gfCNCPoint4[16844] = {X 523.9193, Y 49.0767, Z -5.5000, A 0.000, B 0.000, C 0.000 }
gfCNCPoint4[16845] = {X 523.4026, Y 49.7085, Z -5.5000, A 0.000, B 0.000, C 0.000 }
gfCNCPoint4[16846] = {X 522.7743, Y 50.2295, Z -5.5000, A 0.000, B 0.000, C 0.000 }
gfCNCPoint4[16847] = {X 522.0579, Y 50.6204, Z -5.5000, A 0.000, B 0.000, C 0.000 }
gfCNCPoint4[16848] = {X 521.2797, Y 50.8666, Z -5.5000, A 0.000, B 0.000, C 0.000 }
gfCNCPoint4[16849] = {X 520.4688, Y 50.9591, Z -5.5000, A 0.000, B 0.000, C 0.000 }
gfCNCPoint4[16850] = {X 519.7998, Y 50.9591, Z -5.5000, A 0.000, B 0.000, C 0.000 }
gfCNCPoint4[16851] = {X 518.8919, Y 50.8568, Z -5.5000, A 0.000, B 0.000, C 0.000 }
gfCNCPoint4[16852] = {X 518.0295, Y 50.5551, Z -5.5000, A 0.000, B 0.000, C 0.000 }
gfCNCPoint4[16853] = {X 517.2559, Y 50.0690, Z -5.5000, A 0.000, B 0.000, C 0.000 }
gfCNCPoint4[16854] = {X 516.6099, Y 49.4230, Z -5.5000, A 0.000, B 0.000, C 0.000 }
gfCNCPoint4[16855] = {X 516.1238, Y 48.6494, Z -5.5000, A 0.000, B 0.000, C 0.000 }
gfCNCPoint4[16856] = {X 515.8221, Y 47.7870, Z -5.5000, A 0.000, B 0.000, C 0.000 }
gfCNCPoint4[16857] = {X 515.7198, Y 46.8791, Z -5.5000, A 0.000, B 0.000, C 0.000 }
gfCNCPoint4[16858] = {X 515.7198, Y 39.9011, Z -5.5000, A 0.000, B 0.000, C 0.000 }
gfCNCPoint4[16859] = {X 515.8209, Y 38.9982, Z -5.5000, A 0.000, B 0.000, C 0.000 }
gfCNCPoint4[16860] = {X 516.1194, Y 38.1401, Z -5.5000, A 0.000, B 0.000, C 0.000 }
gfCNCPoint4[16861] = {X 516.6003, Y 37.3693, Z -5.5000, A 0.000, B 0.000, C 0.000 }
gfCNCPoint4[16862] = {X 517.2399, Y 36.7241, Z -5.5000, A 0.000, B 0.000, C 0.000 }
gfCNCPoint4[16863] = {X 518.0064, Y 36.2364, Z -5.5000, A 0.000, B 0.000, C 0.000 }
gfCNCPoint4[16864] = {X 518.8619, Y 35.9304, Z -5.5000, A 0.000, B 0.000, C 0.000 }
gfCNCPoint4[16865] = {X 519.7638, Y 35.8213, Z -5.5000, A 0.000, B 0.000, C 0.000 }
gfCNCPoint4[16866] = {X 520.5236, Y 35.8215, Z -5.5000, A 0.000, B 0.000, C 0.000 }
gfCNCPoint4[16867] = {X 521.3288, Y 35.9129, Z -5.5000, A 0.000, B 0.000, C 0.000 }
gfCNCPoint4[16868] = {X 522.1000, Y 36.1617, Z -5.5000, A 0.000, B 0.000, C 0.000 }
gfCNCPoint4[16869] = {X 522.8069, Y 36.5579, Z -5.5000, A 0.000, B 0.000, C 0.000 }
gfCNCPoint4[16870] = {X 523.4215, Y 37.0861, Z -5.5000, A 0.000, B 0.000, C 0.000 }
gfCNCPoint4[16871] = {X 523.9196, Y 37.7253, Z -5.5000, A 0.000, B 0.000, C 0.000 }
gfCNCPoint4[16872] = {X 534.8719, Y 37.7258, Z -5.5000, A 0.000, B 0.000, C 0.000 }
gfCNCPoint4[16873] = {X 534.8719, Y 33.7257, Z -5.5000, A 0.000, B 0.000, C 0.000 }
gfCNCPoint4[16874] = {X 529.9775, Y 33.7254, Z -5.5000, A 0.000, B 0.000, C 0.000 }
gfCNCPoint4[16875] = {X 529.9071, Y 33.8366, Z -5.5000, A 0.000, B 0.000, C 0.000 }
gfCNCPoint4[16876] = {X 529.2612, Y 34.5790, Z -5.5000, A 0.000, B 0.000, C 0.000 }
gfCNCPoint4[16877] = {X 528.4563, Y 35.1452, Z -5.5000, A 0.000, B 0.000, C 0.000 }
gfCNCPoint4[16878] = {X 527.5392, Y 35.5023, Z -5.5000, A 0.000, B 0.000, C 0.000 }
gfCNCPoint4[16879] = {X 526.5634, Y 35.6293, Z -5.5000, A 0.000, B 0.000, C 0.000 }
gfCNCPoint4[16880] = {X 525.8868, Y 35.6295, Z -5.5000, A 0.000, B 0.000, C 0.000 }
gfCNCPoint4[16881] = {X 524.9789, Y 35.5272, Z -5.5000, A 0.000, B 0.000, C 0.000 }
gfCNCPoint4[16882] = {X 524.1165, Y 35.2254, Z -5.5000, A 0.000, B 0.000, C 0.000 }
gfCNCPoint4[16883] = {X 523.3429, Y 34.7393, Z -5.5000, A 0.000, B 0.000, C 0.000 }
gfCNCPoint4[16884] = {X 522.6969, Y 34.0933, Z -5.5000, A 0.000, B 0.000, C 0.000 }
gfCNCPoint4[16885] = {X 522.2108, Y 33.3197, Z -5.5000, A 0.000, B 0.000, C 0.000 }
gfCNCPoint4[16886] = {X 521.9091, Y 32.4573, Z -5.5000, A 0.000, B 0.000, C 0.000 }
gfCNCPoint4[16887] = {X 521.8068, Y 31.5495, Z -5.5000, A 0.000, B 0.000, C 0.000 }
gfCNCPoint4[16888] = {X 521.8068, Y 24.5714, Z -5.5000, A 0.000, B 0.000, C 0.000 }
gfCNCPoint4[16889] = {X 521.9079, Y 23.6684, Z -5.5000, A 0.000, B 0.000, C 0.000 }
gfCNCPoint4[16890] = {X 522.2065, Y 22.8102, Z -5.5000, A 0.000, B 0.000, C 0.000 }
gfCNCPoint4[16891] = {X 522.6876, Y 22.0393, Z -5.5000, A 0.000, B 0.000, C 0.000 }
gfCNCPoint4[16892] = {X 523.3273, Y 21.3940, Z -5.5000, A 0.000, B 0.000, C 0.000 }
gfCNCPoint4[16893] = {X 524.0941, Y 20.9064, Z -5.5000, A 0.000, B 0.000, C 0.000 }
gfCNCPoint4[16894] = {X 524.9497, Y 20.6005, Z -5.5000, A 0.000, B 0.000, C 0.000 }
gfCNCPoint4[16895] = {X 525.8518, Y 20.4916, Z -5.5000, A 0.000, B 0.000, C 0.000 }
gfCNCPoint4[16896] = {X 526.5672, Y 20.4916, Z -5.5000, A 0.000, B 0.000, C 0.000 }
gfCNCPoint4[16897] = {X 527.3709, Y 20.5794, Z -5.5000, A 0.000, B 0.000, C 0.000 }
gfCNCPoint4[16898] = {X 528.1415, Y 20.8238, Z -5.5000, A 0.000, B 0.000, C 0.000 }
gfCNCPoint4[16899] = {X 528.8488, Y 21.2155, Z -5.5000, A 0.000, B 0.000, C 0.000 }
gfCNCPoint4[16900] = {X 529.4649, Y 21.7389, Z -5.5000, A 0.000, B 0.000, C 0.000 }
gfCNCPoint4[16901] = {X 529.9658, Y 22.3735, Z -5.5000, A 0.000, B 0.000, C 0.000 }
gfCNCPoint4[16902] = {X 534.8719, Y 22.3737, Z -5.5000, A 0.000, B 0.000, C 0.000 }
gfCNCPoint4[16903] = {X 534.8719, Y 19.4621, Z -5.5000, A 0.000, B 0.000, C 0.000 }
gfCNCPoint4[16904] = {X 524.0609, Y 19.4619, Z -5.5000, A 0.000, B 0.000, C 0.000 }
gfCNCPoint4[16905] = {X 524.0087, Y 19.5442, Z -5.5000, A 0.000, B 0.000, C 0.000 }
gfCNCPoint4[16906] = {X 523.5061, Y 20.1604, Z -5.5000, A 0.000, B 0.000, C 0.000 }
gfCNCPoint4[16907] = {X 522.8935, Y 20.6674, Z -5.5000, A 0.000, B 0.000, C 0.000 }
gfCNCPoint4[16908] = {X 522.1942, Y 21.0459, Z -5.5000, A 0.000, B 0.000, C 0.000 }
gfCNCPoint4[16909] = {X 521.4348, Y 21.2816, Z -5.5000, A 0.000, B 0.000, C 0.000 }
gfCNCPoint4[16910] = {X 520.6440, Y 21.3656, Z -5.5000, A 0.000, B 0.000, C 0.000 }
gfCNCPoint4[16911] = {X 519.9691, Y 21.3657, Z -5.5000, A 0.000, B 0.000, C 0.000 }
gfCNCPoint4[16912] = {X 519.0612, Y 21.2634, Z -5.5000, A 0.000, B 0.000, C 0.000 }
gfCNCPoint4[16913] = {X 518.1989, Y 20.9617, Z -5.5000, A 0.000, B 0.000, C 0.000 }
gfCNCPoint4[16914] = {X 517.4253, Y 20.4756, Z -5.5000, A 0.000, B 0.000, C 0.000 }
gfCNCPoint4[16915] = {X 516.7792, Y 19.8296, Z -5.5000, A 0.000, B 0.000, C 0.000 }
gfCNCPoint4[16916] = {X 516.2932, Y 19.0560, Z -5.5000, A 0.000, B 0.000, C 0.000 }
gfCNCPoint4[16917] = {X 515.9914, Y 18.1936, Z -5.5000, A 0.000, B 0.000, C 0.000 }
gfCNCPoint4[16918] = {X 515.8891, Y 17.2857, Z -5.5000, A 0.000, B 0.000, C 0.000 }
gfCNCPoint4[16919] = {X 515.8891, Y 10.3077, Z -5.5000, A 0.000, B 0.000, C 0.000 }
gfCNCPoint4[16920] = {X 515.9902, Y 9.4050, Z -5.5000, A 0.000, B 0.000, C 0.000 }
gfCNCPoint4[16921] = {X 516.2885, Y 8.5471, Z -5.5000, A 0.000, B 0.000, C 0.000 }
gfCNCPoint4[16922] = {X 516.7693, Y 7.7764, Z -5.5000, A 0.000, B 0.000, C 0.000 }
gfCNCPoint4[16923] = {X 517.4086, Y 7.1312, Z -5.5000, A 0.000, B 0.000, C 0.000 }
gfCNCPoint4[16924] = {X 518.1749, Y 6.6434, Z -5.5000, A 0.000, B 0.000, C 0.000 }
gfCNCPoint4[16925] = {X 519.0301, Y 6.3372, Z -5.5000, A 0.000, B 0.000, C 0.000 }
gfCNCPoint4[16926] = {X 519.9318, Y 6.2279, Z -5.5000, A 0.000, B 0.000, C 0.000 }
gfCNCPoint4[16927] = {X 520.6480, Y 6.2279, Z -5.5000, A 0.000, B 0.000, C 0.000 }
gfCNCPoint4[16928] = {X 521.4520, Y 6.3154, Z -5.5000, A 0.000, B 0.000, C 0.000 }
gfCNCPoint4[16929] = {X 522.2230, Y 6.5597, Z -5.5000, A 0.000, B 0.000, C 0.000 }
gfCNCPoint4[16930] = {X 522.9306, Y 6.9514, Z -5.5000, A 0.000, B 0.000, C 0.000 }
gfCNCPoint4[16931] = {X 523.5471, Y 7.4750, Z -5.5000, A 0.000, B 0.000, C 0.000 }
gfCNCPoint4[16932] = {X 524.0482, Y 8.1098, Z -5.5000, A 0.000, B 0.000, C 0.000 }
gfCNCPoint4[16933] = {X 533.9635, Y 8.1100, Z -5.5000, A 0.000, B 0.000, C 0.000 }
gfCNCPoint4[16934] = {X 533.9636, Y 4.1100, Z -5.5000, A 0.000, B 0.000, C 0.000 }
gfCNCPoint4[16935] = {X 533.9635, Y 8.1900, Z -5.5000, A 0.000, B 0.000, C 0.000 }
gfCNCPoint4[16936] = {X 543.7544, Y 8.1902, Z -5.5000, A 0.000, B 0.000, C 0.000 }
gfCNCPoint4[16937] = {X 544.6628, Y 8.2686, Z -5.5000, A 0.000, B 0.000, C 0.000 }
gfCNCPoint4[16938] = {X 545.5299, Y 8.5504, Z -5.5000, A 0.000, B 0.000, C 0.000 }
gfCNCPoint4[16939] = {X 546.3109, Y 9.0210, Z -5.5000, A 0.000, B 0.000, C 0.000 }
gfCNCPoint4[16940] = {X 546.9651, Y 9.6561, Z -5.5000, A 0.000, B 0.000, C 0.000 }
gfCNCPoint4[16941] = {X 547.4587, Y 10.4228, Z -5.5000, A 0.000, B 0.000, C 0.000 }
gfCNCPoint4[16942] = {X 547.7661, Y 11.2812, Z -5.5000, A 0.000, B 0.000, C 0.000 }
gfCNCPoint4[16943] = {X 547.8714, Y 12.1868, Z -5.5000, A 0.000, B 0.000, C 0.000 }
gfCNCPoint4[16944] = {X 547.8712, Y 13.0192, Z -5.5000, A 0.000, B 0.000, C 0.000 }
gfCNCPoint4[16945] = {X 547.7627, Y 13.9043, Z -5.5000, A 0.000, B 0.000, C 0.000 }
gfCNCPoint4[16946] = {X 547.4608, Y 14.7433, Z -5.5000, A 0.000, B 0.000, C 0.000 }
gfCNCPoint4[16947] = {X 546.9806, Y 15.4946, Z -5.5000, A 0.000, B 0.000, C 0.000 }
gfCNCPoint4[16948] = {X 546.3458, Y 16.1209, Z -5.5000, A 0.000, B 0.000, C 0.000 }
gfCNCPoint4[16949] = {X 546.3444, Y 41.0656, Z -5.5000, A 0.000, B 0.000, C 0.000 }
gfCNCPoint4[16950] = {X 546.4832, Y 41.1792, Z -5.5000, A 0.000, B 0.000, C 0.000 }
gfCNCPoint4[16951] = {X 547.0690, Y 41.8056, Z -5.5000, A 0.000, B 0.000, C 0.000 }
gfCNCPoint4[16952] = {X 547.5079, Y 42.5426, Z -5.5000, A 0.000, B 0.000, C 0.000 }
gfCNCPoint4[16953] = {X 547.7795, Y 43.3561, Z -5.5000, A 0.000, B 0.000, C 0.000 }
gfCNCPoint4[16954] = {X 547.8714, Y 44.2089, Z -5.5000, A 0.000, B 0.000, C 0.000 }
gfCNCPoint4[16955] = {X 547.8714, Y 45.0000, Z -5.5000, A 0.000, B 0.000, C 0.000 }
gfCNCPoint4[16956] = {X 547.7662, Y 45.9056, Z -5.5000, A 0.000, B 0.000, C 0.000 }
gfCNCPoint4[16957] = {X 547.4587, Y 46.7640, Z -5.5000, A 0.000, B 0.000, C 0.000 }
gfCNCPoint4[16958] = {X 546.9651, Y 47.5306, Z -5.5000, A 0.000, B 0.000, C 0.000 }
gfCNCPoint4[16959] = {X 546.3109, Y 48.1657, Z -5.5000, A 0.000, B 0.000, C 0.000 }
gfCNCPoint4[16960] = {X 545.5299, Y 48.6363, Z -5.5000, A 0.000, B 0.000, C 0.000 }
gfCNCPoint4[16961] = {X 544.6628, Y 48.9180, Z -5.5000, A 0.000, B 0.000, C 0.000 }
gfCNCPoint4[16962] = {X 543.7544, Y 48.9963, Z -5.5000, A 0.000, B 0.000, C 0.000 }
gfCNCPoint4[16963] = {X 523.8762, Y 48.9967, Z -5.5000, A 0.000, B 0.000, C 0.000 }
gfCNCPoint4[16964] = {X 523.3698, Y 49.6277, Z -5.5000, A 0.000, B 0.000, C 0.000 }
gfCNCPoint4[16965] = {X 522.7508, Y 50.1487, Z -5.5000, A 0.000, B 0.000, C 0.000 }
gfCNCPoint4[16966] = {X 522.0425, Y 50.5399, Z -5.5000, A 0.000, B 0.000, C 0.000 }
gfCNCPoint4[16967] = {X 521.2719, Y 50.7865, Z -5.5000, A 0.000, B 0.000, C 0.000 }
gfCNCPoint4[16968] = {X 520.4681, Y 50.8791, Z -5.5000, A 0.000, B 0.000, C 0.000 }
gfCNCPoint4[16969] = {X 519.7998, Y 50.8791, Z -5.5000, A 0.000, B 0.000, C 0.000 }
gfCNCPoint4[16970] = {X 518.9097, Y 50.7788, Z -5.5000, A 0.000, B 0.000, C 0.000 }
gfCNCPoint4[16971] = {X 518.0642, Y 50.4830, Z -5.5000, A 0.000, B 0.000, C 0.000 }
gfCNCPoint4[16972] = {X 517.3058, Y 50.0064, Z -5.5000, A 0.000, B 0.000, C 0.000 }
gfCNCPoint4[16973] = {X 516.6724, Y 49.3731, Z -5.5000, A 0.000, B 0.000, C 0.000 }
gfCNCPoint4[16974] = {X 516.1959, Y 48.6147, Z -5.5000, A 0.000, B 0.000, C 0.000 }
gfCNCPoint4[16975] = {X 515.9001, Y 47.7692, Z -5.5000, A 0.000, B 0.000, C 0.000 }
gfCNCPoint4[16976] = {X 515.7998, Y 46.8791, Z -5.5000, A 0.000, B 0.000, C 0.000 }
gfCNCPoint4[16977] = {X 515.7998, Y 39.9011, Z -5.5000, A 0.000, B 0.000, C 0.000 }
gfCNCPoint4[16978] = {X 515.9001, Y 39.0110, Z -5.5000, A 0.000, B 0.000, C 0.000 }
gfCNCPoint4[16979] = {X 516.1959, Y 38.1655, Z -5.5000, A 0.000, B 0.000, C 0.000 }
gfCNCPoint4[16980] = {X 516.6725, Y 37.4071, Z -5.5000, A 0.000, B 0.000, C 0.000 }
gfCNCPoint4[16981] = {X 517.3058, Y 36.7738, Z -5.5000, A 0.000, B 0.000, C 0.000 }
gfCNCPoint4[16982] = {X 518.0643, Y 36.2972, Z -5.5000, A 0.000, B 0.000, C 0.000 }
gfCNCPoint4[16983] = {X 518.9097, Y 36.0014, Z -5.5000, A 0.000, B 0.000, C 0.000 }
gfCNCPoint4[16984] = {X 519.7998, Y 35.9011, Z -5.5000, A 0.000, B 0.000, C 0.000 }
gfCNCPoint4[16985] = {X 520.5225, Y 35.9015, Z -5.5000, A 0.000, B 0.000, C 0.000 }
gfCNCPoint4[16986] = {X 521.3205, Y 35.9930, Z -5.5000, A 0.000, B 0.000, C 0.000 }
gfCNCPoint4[16987] = {X 522.0842, Y 36.2421, Z -5.5000, A 0.000, B 0.000, C 0.000 }
gfCNCPoint4[16988] = {X 522.7826, Y 36.6387, Z -5.5000, A 0.000, B 0.000, C 0.000 }
gfCNCPoint4[16989] = {X 523.3878, Y 37.1669, Z -5.5000, A 0.000, B 0.000, C 0.000 }
gfCNCPoint4[16990] = {X 523.8752, Y 37.8053, Z -5.5000, A 0.000, B 0.000, C 0.000 }
gfCNCPoint4[16991] = {X 534.9519, Y 37.8058, Z -5.5000, A 0.000, B 0.000, C 0.000 }
gfCNCPoint4[16992] = {X 534.9519, Y 34.0457, Z -5.5000, A 0.000, B 0.000, C 0.000 }
gfCNCPoint4[16993] = {X 534.9521, Y 33.6457, Z -5.5000, A 0.000, B 0.000, C 0.000 }
gfCNCPoint4[16994] = {X 529.9335, Y 33.6454, Z -5.5000, A 0.000, B 0.000, C 0.000 }
gfCNCPoint4[16995] = {X 529.8226, Y 33.8185, Z -5.5000, A 0.000, B 0.000, C 0.000 }
gfCNCPoint4[16996] = {X 529.1831, Y 34.5416, Z -5.5000, A 0.000, B 0.000, C 0.000 }
gfCNCPoint4[16997] = {X 528.3890, Y 35.0904, Z -5.5000, A 0.000, B 0.000, C 0.000 }
gfCNCPoint4[16998] = {X 527.4865, Y 35.4330, Z -5.5000, A 0.000, B 0.000, C 0.000 }
gfCNCPoint4[16999] = {X 526.5283, Y 35.5495, Z -5.5000, A 0.000, B 0.000, C 0.000 }
gfCNCPoint4[17000] = {X 525.8868, Y 35.5495, Z -5.5000, A 0.000, B 0.000, C 0.000 }
gfCNCPoint4[17001] = {X 524.9967, Y 35.4492, Z -5.5000, A 0.000, B 0.000, C 0.000 }
gfCNCPoint4[17002] = {X 524.1512, Y 35.1533, Z -5.5000, A 0.000, B 0.000, C 0.000 }
gfCNCPoint4[17003] = {X 523.3928, Y 34.6768, Z -5.5000, A 0.000, B 0.000, C 0.000 }
gfCNCPoint4[17004] = {X 522.7594, Y 34.0434, Z -5.5000, A 0.000, B 0.000, C 0.000 }
gfCNCPoint4[17005] = {X 522.2829, Y 33.2850, Z -5.5000, A 0.000, B 0.000, C 0.000 }
gfCNCPoint4[17006] = {X 521.9870, Y 32.4395, Z -5.5000, A 0.000, B 0.000, C 0.000 }
gfCNCPoint4[17007] = {X 521.8868, Y 31.5495, Z -5.5000, A 0.000, B 0.000, C 0.000 }
gfCNCPoint4[17008] = {X 521.8868, Y 24.5714, Z -5.5000, A 0.000, B 0.000, C 0.000 }
gfCNCPoint4[17009] = {X 521.9870, Y 23.6813, Z -5.5000, A 0.000, B 0.000, C 0.000 }
gfCNCPoint4[17010] = {X 522.2829, Y 22.8359, Z -5.5000, A 0.000, B 0.000, C 0.000 }
gfCNCPoint4[17011] = {X 522.7594, Y 22.0775, Z -5.5000, A 0.000, B 0.000, C 0.000 }
gfCNCPoint4[17012] = {X 523.3928, Y 21.4441, Z -5.5000, A 0.000, B 0.000, C 0.000 }
gfCNCPoint4[17013] = {X 524.1512, Y 20.9675, Z -5.5000, A 0.000, B 0.000, C 0.000 }
gfCNCPoint4[17014] = {X 524.9967, Y 20.6717, Z -5.5000, A 0.000, B 0.000, C 0.000 }
gfCNCPoint4[17015] = {X 525.8868, Y 20.5714, Z -5.5000, A 0.000, B 0.000, C 0.000 }
gfCNCPoint4[17016] = {X 526.5664, Y 20.5716, Z -5.5000, A 0.000, B 0.000, C 0.000 }
gfCNCPoint4[17017] = {X 527.3629, Y 20.6594, Z -5.5000, A 0.000, B 0.000, C 0.000 }
gfCNCPoint4[17018] = {X 528.1259, Y 20.9043, Z -5.5000, A 0.000, B 0.000, C 0.000 }
gfCNCPoint4[17019] = {X 528.8248, Y 21.2962, Z -5.5000, A 0.000, B 0.000, C 0.000 }
gfCNCPoint4[17020] = {X 529.4315, Y 21.8197, Z -5.5000, A 0.000, B 0.000, C 0.000 }
gfCNCPoint4[17021] = {X 529.9217, Y 22.4535, Z -5.5000, A 0.000, B 0.000, C 0.000 }
gfCNCPoint4[17022] = {X 534.9519, Y 22.4537, Z -5.5000, A 0.000, B 0.000, C 0.000 }
gfCNCPoint4[17023] = {X 534.9519, Y 19.7821, Z -5.5000, A 0.000, B 0.000, C 0.000 }
gfCNCPoint4[17024] = {X 534.9522, Y 19.3821, Z -5.5000, A 0.000, B 0.000, C 0.000 }
gfCNCPoint4[17025] = {X 524.0169, Y 19.3819, Z -5.5000, A 0.000, B 0.000, C 0.000 }
gfCNCPoint4[17026] = {X 523.9048, Y 19.5550, Z -5.5000, A 0.000, B 0.000, C 0.000 }
gfCNCPoint4[17027] = {X 523.2653, Y 20.2779, Z -5.5000, A 0.000, B 0.000, C 0.000 }
gfCNCPoint4[17028] = {X 522.4713, Y 20.8267, Z -5.5000, A 0.000, B 0.000, C 0.000 }
gfCNCPoint4[17029] = {X 521.5689, Y 21.1693, Z -5.5000, A 0.000, B 0.000, C 0.000 }
gfCNCPoint4[17030] = {X 520.6107, Y 21.2857, Z -5.5000, A 0.000, B 0.000, C 0.000 }
gfCNCPoint4[17031] = {X 519.9691, Y 21.2857, Z -5.5000, A 0.000, B 0.000, C 0.000 }
gfCNCPoint4[17032] = {X 519.0790, Y 21.1854, Z -5.5000, A 0.000, B 0.000, C 0.000 }
gfCNCPoint4[17033] = {X 518.2336, Y 20.8896, Z -5.5000, A 0.000, B 0.000, C 0.000 }
gfCNCPoint4[17034] = {X 517.4751, Y 20.4130, Z -5.5000, A 0.000, B 0.000, C 0.000 }
gfCNCPoint4[17035] = {X 516.8418, Y 19.7797, Z -5.5000, A 0.000, B 0.000, C 0.000 }
gfCNCPoint4[17036] = {X 516.3652, Y 19.0212, Z -5.5000, A 0.000, B 0.000, C 0.000 }
gfCNCPoint4[17037] = {X 516.0694, Y 18.1758, Z -5.5000, A 0.000, B 0.000, C 0.000 }
gfCNCPoint4[17038] = {X 515.9691, Y 17.2857, Z -5.5000, A 0.000, B 0.000, C 0.000 }
gfCNCPoint4[17039] = {X 515.9691, Y 10.3077, Z -5.5000, A 0.000, B 0.000, C 0.000 }
gfCNCPoint4[17040] = {X 516.0694, Y 9.4176, Z -5.5000, A 0.000, B 0.000, C 0.000 }
gfCNCPoint4[17041] = {X 516.3652, Y 8.5721, Z -5.5000, A 0.000, B 0.000, C 0.000 }
gfCNCPoint4[17042] = {X 516.8418, Y 7.8137, Z -5.5000, A 0.000, B 0.000, C 0.000 }
gfCNCPoint4[17043] = {X 517.4752, Y 7.1803, Z -5.5000, A 0.000, B 0.000, C 0.000 }
gfCNCPoint4[17044] = {X 518.2336, Y 6.7038, Z -5.5000, A 0.000, B 0.000, C 0.000 }
gfCNCPoint4[17045] = {X 519.0791, Y 6.4080, Z -5.5000, A 0.000, B 0.000, C 0.000 }
gfCNCPoint4[17046] = {X 519.9692, Y 6.3077, Z -5.5000, A 0.000, B 0.000, C 0.000 }
gfCNCPoint4[17047] = {X 520.6472, Y 6.3079, Z -5.5000, A 0.000, B 0.000, C 0.000 }
gfCNCPoint4[17048] = {X 521.4441, Y 6.3955, Z -5.5000, A 0.000, B 0.000, C 0.000 }
gfCNCPoint4[17049] = {X 522.2074, Y 6.6402, Z -5.5000, A 0.000, B 0.000, C 0.000 }
gfCNCPoint4[17050] = {X 522.9066, Y 7.0322, Z -5.5000, A 0.000, B 0.000, C 0.000 }
gfCNCPoint4[17051] = {X 523.5137, Y 7.5557, Z -5.5000, A 0.000, B 0.000, C 0.000 }
gfCNCPoint4[17052] = {X 524.0041, Y 8.1898, Z -5.5000, A 0.000, B 0.000, C 0.000 }
gfCNCPoint4[17053] = {X 533.9635, Y 8.1900, Z -5.5000, A 0.000, B 0.000, C 0.000 }
gfCNCPoint4[17054] = {X 533.9636, Y 4.1100, Z -5.5000, A 0.000, B 0.000, C 0.000 }
gfCNCPoint4[17055] = {X 533.9636, Y 4.1100, Z -2.5000, A 0.000, B 0.000, C 0.000 }
gfCNCPoint4[17056] = {X 533.9636, Y 4.1100, Z 11.0000, A 0.000, B 0.000, C 0.000 }
gfCNCPoint4[17057] = {X 419.6144, Y 26.5282, Z 11.0000, A 0.000, B 0.000, C 0.000 }
gfCNCPoint4[17058] = {X 419.6144, Y 26.5282, Z -2.5000, A 0.000, B 0.000, C 0.000 }
gfCNCPoint4[17059] = {X 419.6144, Y 26.5282, Z -5.5000, A 0.000, B 0.000, C 0.000 }
gfCNCPoint4[17060] = {X 416.1509, Y 24.3717, Z -5.5000, A 0.000, B 0.000, C 0.000 }
gfCNCPoint4[17061] = {X 411.5473, Y 31.7652, Z -5.5000, A 0.000, B 0.000, C 0.000 }
gfCNCPoint4[17062] = {X 411.5479, Y 40.8978, Z -5.5000, A 0.000, B 0.000, C 0.000 }
gfCNCPoint4[17063] = {X 412.1861, Y 41.5837, Z -5.5000, A 0.000, B 0.000, C 0.000 }
gfCNCPoint4[17064] = {X 412.6662, Y 42.3882, Z -5.5000, A 0.000, B 0.000, C 0.000 }
gfCNCPoint4[17065] = {X 412.9668, Y 43.2755, Z -5.5000, A 0.000, B 0.000, C 0.000 }
gfCNCPoint4[17066] = {X 413.0747, Y 44.2062, Z -5.5000, A 0.000, B 0.000, C 0.000 }
gfCNCPoint4[17067] = {X 413.0747, Y 45.0002, Z -5.5000, A 0.000, B 0.000, C 0.000 }
gfCNCPoint4[17068] = {X 412.9663, Y 45.9614, Z -5.5000, A 0.000, B 0.000, C 0.000 }
gfCNCPoint4[17069] = {X 412.6468, Y 46.8745, Z -5.5000, A 0.000, B 0.000, C 0.000 }
gfCNCPoint4[17070] = {X 412.1321, Y 47.6936, Z -5.5000, A 0.000, B 0.000, C 0.000 }
gfCNCPoint4[17071] = {X 411.4481, Y 48.3776, Z -5.5000, A 0.000, B 0.000, C 0.000 }
gfCNCPoint4[17072] = {X 410.6290, Y 48.8922, Z -5.5000, A 0.000, B 0.000, C 0.000 }
gfCNCPoint4[17073] = {X 409.7159, Y 49.2117, Z -5.5000, A 0.000, B 0.000, C 0.000 }
gfCNCPoint4[17074] = {X 408.7547, Y 49.3200, Z -5.5000, A 0.000, B 0.000, C 0.000 }
gfCNCPoint4[17075] = {X 402.3112, Y 49.3200, Z -5.5000, A 0.000, B 0.000, C 0.000 }
gfCNCPoint4[17076] = {X 401.3546, Y 49.2127, Z -5.5000, A 0.000, B 0.000, C 0.000 }
gfCNCPoint4[17077] = {X 400.4455, Y 48.8963, Z -5.5000, A 0.000, B 0.000, C 0.000 }
gfCNCPoint4[17078] = {X 399.6290, Y 48.3864, Z -5.5000, A 0.000, B 0.000, C 0.000 }
gfCNCPoint4[17079] = {X 398.9457, Y 47.7084, Z -5.5000, A 0.000, B 0.000, C 0.000 }
gfCNCPoint4[17080] = {X 398.4295, Y 46.8959, Z -5.5000, A 0.000, B 0.000, C 0.000 }
gfCNCPoint4[17081] = {X 398.1060, Y 45.9892, Z -5.5000, A 0.000, B 0.000, C 0.000 }
gfCNCPoint4[17082] = {X 397.9913, Y 45.0335, Z -5.5000, A 0.000, B 0.000, C 0.000 }
gfCNCPoint4[17083] = {X 397.9916, Y 44.1528, Z -5.5000, A 0.000, B 0.000, C 0.000 }
gfCNCPoint4[17084] = {X 398.1015, Y 43.2391, Z -5.5000, A 0.000, B 0.000, C 0.000 }
gfCNCPoint4[17085] = {X 398.4024, Y 42.3694, Z -5.5000, A 0.000, B 0.000, C 0.000 }
gfCNCPoint4[17086] = {X 398.8807, Y 41.5832, Z -5.5000, A 0.000, B 0.000, C 0.000 }
gfCNCPoint4[17087] = {X 399.5147, Y 40.9161, Z -5.5000, A 0.000, B 0.000, C 0.000 }
gfCNCPoint4[17088] = {X 399.4729, Y 31.6010, Z -5.5000, A 0.000, B 0.000, C 0.000 }
gfCNCPoint4[17089] = {X 393.5178, Y 21.2453, Z -5.5000, A 0.000, B 0.000, C 0.000 }
gfCNCPoint4[17090] = {X 392.6297, Y 19.7345, Z -5.5000, A 0.000, B 0.000, C 0.000 }
gfCNCPoint4[17091] = {X 391.7131, Y 18.2409, Z -5.5000, A 0.000, B 0.000, C 0.000 }
gfCNCPoint4[17092] = {X 391.2305, Y 17.5698, Z -5.5000, A 0.000, B 0.000, C 0.000 }
gfCNCPoint4[17093] = {X 390.6669, Y 16.9652, Z -5.5000, A 0.000, B 0.000, C 0.000 }
gfCNCPoint4[17094] = {X 389.7902, Y 16.4728, Z -5.5000, A 0.000, B 0.000, C 0.000 }
gfCNCPoint4[17095] = {X 389.0510, Y 15.7911, Z -5.5000, A 0.000, B 0.000, C 0.000 }
gfCNCPoint4[17096] = {X 388.4895, Y 14.9569, Z -5.5000, A 0.000, B 0.000, C 0.000 }
gfCNCPoint4[17097] = {X 388.1361, Y 14.0156, Z -5.5000, A 0.000, B 0.000, C 0.000 }
gfCNCPoint4[17098] = {X 388.0098, Y 13.0180, Z -5.5000, A 0.000, B 0.000, C 0.000 }
gfCNCPoint4[17099] = {X 388.0096, Y 12.1868, Z -5.5000, A 0.000, B 0.000, C 0.000 }
gfCNCPoint4[17100] = {X 388.1179, Y 11.2255, Z -5.5000, A 0.000, B 0.000, C 0.000 }
gfCNCPoint4[17101] = {X 388.4374, Y 10.3125, Z -5.5000, A 0.000, B 0.000, C 0.000 }
gfCNCPoint4[17102] = {X 388.9521, Y 9.4933, Z -5.5000, A 0.000, B 0.000, C 0.000 }
gfCNCPoint4[17103] = {X 389.6361, Y 8.8093, Z -5.5000, A 0.000, B 0.000, C 0.000 }
gfCNCPoint4[17104] = {X 390.4552, Y 8.2946, Z -5.5000, A 0.000, B 0.000, C 0.000 }
gfCNCPoint4[17105] = {X 391.3683, Y 7.9751, Z -5.5000, A 0.000, B 0.000, C 0.000 }
gfCNCPoint4[17106] = {X 392.3296, Y 7.8668, Z -5.5000, A 0.000, B 0.000, C 0.000 }
gfCNCPoint4[17107] = {X 399.1118, Y 7.8668, Z -5.5000, A 0.000, B 0.000, C 0.000 }
gfCNCPoint4[17108] = {X 400.0730, Y 7.9751, Z -5.5000, A 0.000, B 0.000, C 0.000 }
gfCNCPoint4[17109] = {X 400.9861, Y 8.2946, Z -5.5000, A 0.000, B 0.000, C 0.000 }
gfCNCPoint4[17110] = {X 401.8052, Y 8.8093, Z -5.5000, A 0.000, B 0.000, C 0.000 }
gfCNCPoint4[17111] = {X 402.4893, Y 9.4933, Z -5.5000, A 0.000, B 0.000, C 0.000 }
gfCNCPoint4[17112] = {X 403.0039, Y 10.3124, Z -5.5000, A 0.000, B 0.000, C 0.000 }
gfCNCPoint4[17113] = {X 403.3234, Y 11.2255, Z -5.5000, A 0.000, B 0.000, C 0.000 }
gfCNCPoint4[17114] = {X 403.4318, Y 12.1868, Z -5.5000, A 0.000, B 0.000, C 0.000 }
gfCNCPoint4[17115] = {X 403.4318, Y 12.9782, Z -5.5000, A 0.000, B 0.000, C 0.000 }
gfCNCPoint4[17116] = {X 403.3293, Y 13.9134, Z -5.5000, A 0.000, B 0.000, C 0.000 }
gfCNCPoint4[17117] = {X 403.0267, Y 14.8043, Z -5.5000, A 0.000, B 0.000, C 0.000 }
gfCNCPoint4[17118] = {X 405.3561, Y 18.8228, Z -5.5000, A 0.000, B 0.000, C 0.000 }
gfCNCPoint4[17119] = {X 407.8733, Y 14.7536, Z -5.5000, A 0.000, B 0.000, C 0.000 }
gfCNCPoint4[17120] = {X 407.5920, Y 13.9042, Z -5.5000, A 0.000, B 0.000, C 0.000 }
gfCNCPoint4[17121] = {X 407.4917, Y 13.0151, Z -5.5000, A 0.000, B 0.000, C 0.000 }
gfCNCPoint4[17122] = {X 407.4915, Y 12.1868, Z -5.5000, A 0.000, B 0.000, C 0.000 }
gfCNCPoint4[17123] = {X 407.5999, Y 11.2255, Z -5.5000, A 0.000, B 0.000, C 0.000 }
gfCNCPoint4[17124] = {X 407.9194, Y 10.3124, Z -5.5000, A 0.000, B 0.000, C 0.000 }
gfCNCPoint4[17125] = {X 408.4340, Y 9.4933, Z -5.5000, A 0.000, B 0.000, C 0.000 }
gfCNCPoint4[17126] = {X 409.1181, Y 8.8093, Z -5.5000, A 0.000, B 0.000, C 0.000 }
gfCNCPoint4[17127] = {X 409.9372, Y 8.2946, Z -5.5000, A 0.000, B 0.000, C 0.000 }
gfCNCPoint4[17128] = {X 410.8502, Y 7.9751, Z -5.5000, A 0.000, B 0.000, C 0.000 }
gfCNCPoint4[17129] = {X 411.8115, Y 7.8668, Z -5.5000, A 0.000, B 0.000, C 0.000 }
gfCNCPoint4[17130] = {X 419.3245, Y 7.8668, Z -5.5000, A 0.000, B 0.000, C 0.000 }
gfCNCPoint4[17131] = {X 420.2858, Y 7.9751, Z -5.5000, A 0.000, B 0.000, C 0.000 }
gfCNCPoint4[17132] = {X 421.1988, Y 8.2946, Z -5.5000, A 0.000, B 0.000, C 0.000 }
gfCNCPoint4[17133] = {X 422.0179, Y 8.8093, Z -5.5000, A 0.000, B 0.000, C 0.000 }
gfCNCPoint4[17134] = {X 422.7020, Y 9.4933, Z -5.5000, A 0.000, B 0.000, C 0.000 }
gfCNCPoint4[17135] = {X 423.2166, Y 10.3124, Z -5.5000, A 0.000, B 0.000, C 0.000 }
gfCNCPoint4[17136] = {X 423.5361, Y 11.2255, Z -5.5000, A 0.000, B 0.000, C 0.000 }
gfCNCPoint4[17137] = {X 423.6445, Y 12.1868, Z -5.5000, A 0.000, B 0.000, C 0.000 }
gfCNCPoint4[17138] = {X 423.6445, Y 12.9802, Z -5.5000, A 0.000, B 0.000, C 0.000 }
gfCNCPoint4[17139] = {X 423.5517, Y 13.8468, Z -5.5000, A 0.000, B 0.000, C 0.000 }
gfCNCPoint4[17140] = {X 423.2893, Y 14.6779, Z -5.5000, A 0.000, B 0.000, C 0.000 }
gfCNCPoint4[17141] = {X 422.8676, Y 15.4406, Z -5.5000, A 0.000, B 0.000, C 0.000 }
gfCNCPoint4[17142] = {X 422.3034, Y 16.1048, Z -5.5000, A 0.000, B 0.000, C 0.000 }
gfCNCPoint4[17143] = {X 421.6189, Y 16.6442, Z -5.5000, A 0.000, B 0.000, C 0.000 }
gfCNCPoint4[17144] = {X 420.8412, Y 17.0376, Z -5.5000, A 0.000, B 0.000, C 0.000 }
gfCNCPoint4[17145] = {X 420.1248, Y 18.0010, Z -5.5000, A 0.000, B 0.000, C 0.000 }
gfCNCPoint4[17146] = {X 419.4766, Y 19.0115, Z -5.5000, A 0.000, B 0.000, C 0.000 }
gfCNCPoint4[17147] = {X 417.9942, Y 21.4114, Z -5.5000, A 0.000, B 0.000, C 0.000 }
gfCNCPoint4[17148] = {X 416.1509, Y 24.3717, Z -5.5000, A 0.000, B 0.000, C 0.000 }
gfCNCPoint4[17149] = {X 419.5465, Y 26.4860, Z -5.5000, A 0.000, B 0.000, C 0.000 }
gfCNCPoint4[17150] = {X 416.0830, Y 24.3294, Z -5.5000, A 0.000, B 0.000, C 0.000 }
gfCNCPoint4[17151] = {X 411.4673, Y 31.7423, Z -5.5000, A 0.000, B 0.000, C 0.000 }
gfCNCPoint4[17152] = {X 411.4679, Y 40.9345, Z -5.5000, A 0.000, B 0.000, C 0.000 }
gfCNCPoint4[17153] = {X 412.1057, Y 41.6100, Z -5.5000, A 0.000, B 0.000, C 0.000 }
gfCNCPoint4[17154] = {X 412.5859, Y 42.4052, Z -5.5000, A 0.000, B 0.000, C 0.000 }
gfCNCPoint4[17155] = {X 412.8868, Y 43.2842, Z -5.5000, A 0.000, B 0.000, C 0.000 }
gfCNCPoint4[17156] = {X 412.9947, Y 44.2069, Z -5.5000, A 0.000, B 0.000, C 0.000 }
gfCNCPoint4[17157] = {X 412.9947, Y 45.0002, Z -5.5000, A 0.000, B 0.000, C 0.000 }
gfCNCPoint4[17158] = {X 412.8883, Y 45.9436, Z -5.5000, A 0.000, B 0.000, C 0.000 }
gfCNCPoint4[17159] = {X 412.5747, Y 46.8398, Z -5.5000, A 0.000, B 0.000, C 0.000 }
gfCNCPoint4[17160] = {X 412.0696, Y 47.6437, Z -5.5000, A 0.000, B 0.000, C 0.000 }
gfCNCPoint4[17161] = {X 411.3982, Y 48.3150, Z -5.5000, A 0.000, B 0.000, C 0.000 }
gfCNCPoint4[17162] = {X 410.5943, Y 48.8201, Z -5.5000, A 0.000, B 0.000, C 0.000 }
gfCNCPoint4[17163] = {X 409.6981, Y 49.1337, Z -5.5000, A 0.000, B 0.000, C 0.000 }
gfCNCPoint4[17164] = {X 408.7547, Y 49.2400, Z -5.5000, A 0.000, B 0.000, C 0.000 }
gfCNCPoint4[17165] = {X 402.3112, Y 49.2400, Z -5.5000, A 0.000, B 0.000, C 0.000 }
gfCNCPoint4[17166] = {X 401.3723, Y 49.1347, Z -5.5000, A 0.000, B 0.000, C 0.000 }
gfCNCPoint4[17167] = {X 400.4800, Y 48.8242, Z -5.5000, A 0.000, B 0.000, C 0.000 }
gfCNCPoint4[17168] = {X 399.6786, Y 48.3237, Z -5.5000, A 0.000, B 0.000, C 0.000 }
gfCNCPoint4[17169] = {X 399.0080, Y 47.6582, Z -5.5000, A 0.000, B 0.000, C 0.000 }
gfCNCPoint4[17170] = {X 398.5013, Y 46.8608, Z -5.5000, A 0.000, B 0.000, C 0.000 }
gfCNCPoint4[17171] = {X 398.1839, Y 45.9709, Z -5.5000, A 0.000, B 0.000, C 0.000 }
gfCNCPoint4[17172] = {X 398.0713, Y 45.0329, Z -5.5000, A 0.000, B 0.000, C 0.000 }
gfCNCPoint4[17173] = {X 398.0716, Y 44.1538, Z -5.5000, A 0.000, B 0.000, C 0.000 }
gfCNCPoint4[17174] = {X 398.1815, Y 43.2480, Z -5.5000, A 0.000, B 0.000, C 0.000 }
gfCNCPoint4[17175] = {X 398.4827, Y 42.3867, Z -5.5000, A 0.000, B 0.000, C 0.000 }
gfCNCPoint4[17176] = {X 398.9612, Y 41.6098, Z -5.5000, A 0.000, B 0.000, C 0.000 }
gfCNCPoint4[17177] = {X 399.5948, Y 40.9532, Z -5.5000, A 0.000, B 0.000, C 0.000 }
gfCNCPoint4[17178] = {X 399.5528, Y 31.5795, Z -5.5000, A 0.000, B 0.000, C 0.000 }
gfCNCPoint4[17179] = {X 393.5872, Y 21.2054, Z -5.5000, A 0.000, B 0.000, C 0.000 }
gfCNCPoint4[17180] = {X 392.6983, Y 19.6933, Z -5.5000, A 0.000, B 0.000, C 0.000 }
gfCNCPoint4[17181] = {X 391.7809, Y 18.1984, Z -5.5000, A 0.000, B 0.000, C 0.000 }
gfCNCPoint4[17182] = {X 391.2877, Y 17.5134, Z -5.5000, A 0.000, B 0.000, C 0.000 }
gfCNCPoint4[17183] = {X 390.7111, Y 16.8969, Z -5.5000, A 0.000, B 0.000, C 0.000 }
gfCNCPoint4[17184] = {X 389.8466, Y 16.4149, Z -5.5000, A 0.000, B 0.000, C 0.000 }
gfCNCPoint4[17185] = {X 389.1174, Y 15.7456, Z -5.5000, A 0.000, B 0.000, C 0.000 }
gfCNCPoint4[17186] = {X 388.5633, Y 14.9255, Z -5.5000, A 0.000, B 0.000, C 0.000 }
gfCNCPoint4[17187] = {X 388.2144, Y 13.9992, Z -5.5000, A 0.000, B 0.000, C 0.000 }
gfCNCPoint4[17188] = {X 388.0898, Y 13.0173, Z -5.5000, A 0.000, B 0.000, C 0.000 }
gfCNCPoint4[17189] = {X 388.0896, Y 12.1868, Z -5.5000, A 0.000, B 0.000, C 0.000 }
gfCNCPoint4[17190] = {X 388.1959, Y 11.2433, Z -5.5000, A 0.000, B 0.000, C 0.000 }
gfCNCPoint4[17191] = {X 388.5095, Y 10.3472, Z -5.5000, A 0.000, B 0.000, C 0.000 }
gfCNCPoint4[17192] = {X 389.0147, Y 9.5432, Z -5.5000, A 0.000, B 0.000, C 0.000 }
gfCNCPoint4[17193] = {X 389.6860, Y 8.8719, Z -5.5000, A 0.000, B 0.000, C 0.000 }
gfCNCPoint4[17194] = {X 390.4900, Y 8.3667, Z -5.5000, A 0.000, B 0.000, C 0.000 }
gfCNCPoint4[17195] = {X 391.3861, Y 8.0531, Z -5.5000, A 0.000, B 0.000, C 0.000 }
gfCNCPoint4[17196] = {X 392.3296, Y 7.9468, Z -5.5000, A 0.000, B 0.000, C 0.000 }
gfCNCPoint4[17197] = {X 399.1118, Y 7.9468, Z -5.5000, A 0.000, B 0.000, C 0.000 }
gfCNCPoint4[17198] = {X 400.0552, Y 8.0531, Z -5.5000, A 0.000, B 0.000, C 0.000 }
gfCNCPoint4[17199] = {X 400.9514, Y 8.3667, Z -5.5000, A 0.000, B 0.000, C 0.000 }
gfCNCPoint4[17200] = {X 401.7554, Y 8.8718, Z -5.5000, A 0.000, B 0.000, C 0.000 }
gfCNCPoint4[17201] = {X 402.4267, Y 9.5432, Z -5.5000, A 0.000, B 0.000, C 0.000 }
gfCNCPoint4[17202] = {X 402.9319, Y 10.3471, Z -5.5000, A 0.000, B 0.000, C 0.000 }
gfCNCPoint4[17203] = {X 403.2455, Y 11.2433, Z -5.5000, A 0.000, B 0.000, C 0.000 }
gfCNCPoint4[17204] = {X 403.3518, Y 12.1868, Z -5.5000, A 0.000, B 0.000, C 0.000 }
gfCNCPoint4[17205] = {X 403.3518, Y 12.9782, Z -5.5000, A 0.000, B 0.000, C 0.000 }
gfCNCPoint4[17206] = {X 403.2466, Y 13.9164, Z -5.5000, A 0.000, B 0.000, C 0.000 }
gfCNCPoint4[17207] = {X 402.9364, Y 14.8081, Z -5.5000, A 0.000, B 0.000, C 0.000 }
gfCNCPoint4[17208] = {X 405.3539, Y 18.9785, Z -5.5000, A 0.000, B 0.000, C 0.000 }
gfCNCPoint4[17209] = {X 407.9639, Y 14.7593, Z -5.5000, A 0.000, B 0.000, C 0.000 }
gfCNCPoint4[17210] = {X 407.6747, Y 13.9078, Z -5.5000, A 0.000, B 0.000, C 0.000 }
gfCNCPoint4[17211] = {X 407.5717, Y 13.0144, Z -5.5000, A 0.000, B 0.000, C 0.000 }
gfCNCPoint4[17212] = {X 407.5715, Y 12.1868, Z -5.5000, A 0.000, B 0.000, C 0.000 }
gfCNCPoint4[17213] = {X 407.6778, Y 11.2433, Z -5.5000, A 0.000, B 0.000, C 0.000 }
gfCNCPoint4[17214] = {X 407.9914, Y 10.3471, Z -5.5000, A 0.000, B 0.000, C 0.000 }
gfCNCPoint4[17215] = {X 408.4966, Y 9.5432, Z -5.5000, A 0.000, B 0.000, C 0.000 }
gfCNCPoint4[17216] = {X 409.1679, Y 8.8718, Z -5.5000, A 0.000, B 0.000, C 0.000 }
gfCNCPoint4[17217] = {X 409.9719, Y 8.3667, Z -5.5000, A 0.000, B 0.000, C 0.000 }
gfCNCPoint4[17218] = {X 410.8680, Y 8.0531, Z -5.5000, A 0.000, B 0.000, C 0.000 }
gfCNCPoint4[17219] = {X 411.8115, Y 7.9468, Z -5.5000, A 0.000, B 0.000, C 0.000 }
gfCNCPoint4[17220] = {X 419.3245, Y 7.9468, Z -5.5000, A 0.000, B 0.000, C 0.000 }
gfCNCPoint4[17221] = {X 420.2679, Y 8.0531, Z -5.5000, A 0.000, B 0.000, C 0.000 }
gfCNCPoint4[17222] = {X 421.1641, Y 8.3667, Z -5.5000, A 0.000, B 0.000, C 0.000 }
gfCNCPoint4[17223] = {X 421.9681, Y 8.8718, Z -5.5000, A 0.000, B 0.000, C 0.000 }
gfCNCPoint4[17224] = {X 422.6394, Y 9.5432, Z -5.5000, A 0.000, B 0.000, C 0.000 }
gfCNCPoint4[17225] = {X 423.1446, Y 10.3471, Z -5.5000, A 0.000, B 0.000, C 0.000 }
gfCNCPoint4[17226] = {X 423.4582, Y 11.2433, Z -5.5000, A 0.000, B 0.000, C 0.000 }
gfCNCPoint4[17227] = {X 423.5645, Y 12.1868, Z -5.5000, A 0.000, B 0.000, C 0.000 }
gfCNCPoint4[17228] = {X 423.5645, Y 12.9797, Z -5.5000, A 0.000, B 0.000, C 0.000 }
gfCNCPoint4[17229] = {X 423.4726, Y 13.8339, Z -5.5000, A 0.000, B 0.000, C 0.000 }
gfCNCPoint4[17230] = {X 423.2129, Y 14.6529, Z -5.5000, A 0.000, B 0.000, C 0.000 }
gfCNCPoint4[17231] = {X 422.7957, Y 15.4040, Z -5.5000, A 0.000, B 0.000, C 0.000 }
gfCNCPoint4[17232] = {X 422.2375, Y 16.0571, Z -5.5000, A 0.000, B 0.000, C 0.000 }
gfCNCPoint4[17233] = {X 421.5607, Y 16.5864, Z -5.5000, A 0.000, B 0.000, C 0.000 }
gfCNCPoint4[17234] = {X 420.7923, Y 16.9707, Z -5.5000, A 0.000, B 0.000, C 0.000 }
gfCNCPoint4[17235] = {X 420.0654, Y 17.9462, Z -5.5000, A 0.000, B 0.000, C 0.000 }
gfCNCPoint4[17236] = {X 419.4081, Y 18.9700, Z -5.5000, A 0.000, B 0.000, C 0.000 }
gfCNCPoint4[17237] = {X 417.9262, Y 21.3692, Z -5.5000, A 0.000, B 0.000, C 0.000 }
gfCNCPoint4[17238] = {X 416.0830, Y 24.3294, Z -5.5000, A 0.000, B 0.000, C 0.000 }
gfCNCPoint4[17239] = {X 419.4786, Y 26.4437, Z -5.5000, A 0.000, B 0.000, C 0.000 }
gfCNCPoint4[17240] = {X 416.0151, Y 24.2871, Z -5.5000, A 0.000, B 0.000, C 0.000 }
gfCNCPoint4[17241] = {X 411.3873, Y 31.7195, Z -5.5000, A 0.000, B 0.000, C 0.000 }
gfCNCPoint4[17242] = {X 411.3879, Y 40.9715, Z -5.5000, A 0.000, B 0.000, C 0.000 }
gfCNCPoint4[17243] = {X 412.0253, Y 41.6365, Z -5.5000, A 0.000, B 0.000, C 0.000 }
gfCNCPoint4[17244] = {X 412.5056, Y 42.4225, Z -5.5000, A 0.000, B 0.000, C 0.000 }
gfCNCPoint4[17245] = {X 412.8067, Y 43.2929, Z -5.5000, A 0.000, B 0.000, C 0.000 }
gfCNCPoint4[17246] = {X 412.9147, Y 44.2077, Z -5.5000, A 0.000, B 0.000, C 0.000 }
gfCNCPoint4[17247] = {X 412.9147, Y 45.0002, Z -5.5000, A 0.000, B 0.000, C 0.000 }
gfCNCPoint4[17248] = {X 412.8103, Y 45.9258, Z -5.5000, A 0.000, B 0.000, C 0.000 }
gfCNCPoint4[17249] = {X 412.5027, Y 46.8051, Z -5.5000, A 0.000, B 0.000, C 0.000 }
gfCNCPoint4[17250] = {X 412.0070, Y 47.5938, Z -5.5000, A 0.000, B 0.000, C 0.000 }
gfCNCPoint4[17251] = {X 411.3483, Y 48.2525, Z -5.5000, A 0.000, B 0.000, C 0.000 }
gfCNCPoint4[17252] = {X 410.5596, Y 48.7480, Z -5.5000, A 0.000, B 0.000, C 0.000 }
gfCNCPoint4[17253] = {X 409.6803, Y 49.0557, Z -5.5000, A 0.000, B 0.000, C 0.000 }
gfCNCPoint4[17254] = {X 408.7547, Y 49.1600, Z -5.5000, A 0.000, B 0.000, C 0.000 }
gfCNCPoint4[17255] = {X 402.3112, Y 49.1600, Z -5.5000, A 0.000, B 0.000, C 0.000 }
gfCNCPoint4[17256] = {X 401.3900, Y 49.0567, Z -5.5000, A 0.000, B 0.000, C 0.000 }
gfCNCPoint4[17257] = {X 400.5146, Y 48.7520, Z -5.5000, A 0.000, B 0.000, C 0.000 }
gfCNCPoint4[17258] = {X 399.7283, Y 48.2610, Z -5.5000, A 0.000, B 0.000, C 0.000 }
gfCNCPoint4[17259] = {X 399.0703, Y 47.6081, Z -5.5000, A 0.000, B 0.000, C 0.000 }
gfCNCPoint4[17260] = {X 398.5732, Y 46.8257, Z -5.5000, A 0.000, B 0.000, C 0.000 }
gfCNCPoint4[17261] = {X 398.2617, Y 45.9526, Z -5.5000, A 0.000, B 0.000, C 0.000 }
gfCNCPoint4[17262] = {X 398.1513, Y 45.0322, Z -5.5000, A 0.000, B 0.000, C 0.000 }
gfCNCPoint4[17263] = {X 398.1516, Y 44.1549, Z -5.5000, A 0.000, B 0.000, C 0.000 }
gfCNCPoint4[17264] = {X 398.2616, Y 43.2570, Z -5.5000, A 0.000, B 0.000, C 0.000 }
gfCNCPoint4[17265] = {X 398.5630, Y 42.4041, Z -5.5000, A 0.000, B 0.000, C 0.000 }
gfCNCPoint4[17266] = {X 399.0417, Y 41.6366, Z -5.5000, A 0.000, B 0.000, C 0.000 }
gfCNCPoint4[17267] = {X 399.6750, Y 40.9907, Z -5.5000, A 0.000, B 0.000, C 0.000 }
gfCNCPoint4[17268] = {X 399.6327, Y 31.5579, Z -5.5000, A 0.000, B 0.000, C 0.000 }
gfCNCPoint4[17269] = {X 393.6565, Y 21.1656, Z -5.5000, A 0.000, B 0.000, C 0.000 }
gfCNCPoint4[17270] = {X 392.7669, Y 19.6521, Z -5.5000, A 0.000, B 0.000, C 0.000 }
gfCNCPoint4[17271] = {X 391.8486, Y 18.1559, Z -5.5000, A 0.000, B 0.000, C 0.000 }
gfCNCPoint4[17272] = {X 391.3448, Y 17.4569, Z -5.5000, A 0.000, B 0.000, C 0.000 }
gfCNCPoint4[17273] = {X 390.7551, Y 16.8285, Z -5.5000, A 0.000, B 0.000, C 0.000 }
gfCNCPoint4[17274] = {X 389.9029, Y 16.3569, Z -5.5000, A 0.000, B 0.000, C 0.000 }
gfCNCPoint4[17275] = {X 389.1838, Y 15.7000, Z -5.5000, A 0.000, B 0.000, C 0.000 }
gfCNCPoint4[17276] = {X 388.6371, Y 14.8939, Z -5.5000, A 0.000, B 0.000, C 0.000 }
gfCNCPoint4[17277] = {X 388.2928, Y 13.9828, Z -5.5000, A 0.000, B 0.000, C 0.000 }
gfCNCPoint4[17278] = {X 388.1698, Y 13.0166, Z -5.5000, A 0.000, B 0.000, C 0.000 }
gfCNCPoint4[17279] = {X 388.1696, Y 12.1868, Z -5.5000, A 0.000, B 0.000, C 0.000 }
gfCNCPoint4[17280] = {X 388.2739, Y 11.2611, Z -5.5000, A 0.000, B 0.000, C 0.000 }
gfCNCPoint4[17281] = {X 388.5816, Y 10.3819, Z -5.5000, A 0.000, B 0.000, C 0.000 }
gfCNCPoint4[17282] = {X 389.0772, Y 9.5931, Z -5.5000, A 0.000, B 0.000, C 0.000 }
gfCNCPoint4[17283] = {X 389.7359, Y 8.9344, Z -5.5000, A 0.000, B 0.000, C 0.000 }
gfCNCPoint4[17284] = {X 390.5247, Y 8.4388, Z -5.5000, A 0.000, B 0.000, C 0.000 }
gfCNCPoint4[17285] = {X 391.4039, Y 8.1311, Z -5.5000, A 0.000, B 0.000, C 0.000 }
gfCNCPoint4[17286] = {X 392.3296, Y 8.0268, Z -5.5000, A 0.000, B 0.000, C 0.000 }
gfCNCPoint4[17287] = {X 399.1118, Y 8.0268, Z -5.5000, A 0.000, B 0.000, C 0.000 }
gfCNCPoint4[17288] = {X 400.0374, Y 8.1311, Z -5.5000, A 0.000, B 0.000, C 0.000 }
gfCNCPoint4[17289] = {X 400.9167, Y 8.4388, Z -5.5000, A 0.000, B 0.000, C 0.000 }
gfCNCPoint4[17290] = {X 401.7055, Y 8.9344, Z -5.5000, A 0.000, B 0.000, C 0.000 }
gfCNCPoint4[17291] = {X 402.3642, Y 9.5931, Z -5.5000, A 0.000, B 0.000, C 0.000 }
gfCNCPoint4[17292] = {X 402.8598, Y 10.3819, Z -5.5000, A 0.000, B 0.000, C 0.000 }
gfCNCPoint4[17293] = {X 403.1675, Y 11.2611, Z -5.5000, A 0.000, B 0.000, C 0.000 }
gfCNCPoint4[17294] = {X 403.2718, Y 12.1868, Z -5.5000, A 0.000, B 0.000, C 0.000 }
gfCNCPoint4[17295] = {X 403.2718, Y 12.9782, Z -5.5000, A 0.000, B 0.000, C 0.000 }
gfCNCPoint4[17296] = {X 403.1639, Y 13.9192, Z -5.5000, A 0.000, B 0.000, C 0.000 }
gfCNCPoint4[17297] = {X 402.8459, Y 14.8115, Z -5.5000, A 0.000, B 0.000, C 0.000 }
gfCNCPoint4[17298] = {X 405.3517, Y 19.1342, Z -5.5000, A 0.000, B 0.000, C 0.000 }
gfCNCPoint4[17299] = {X 408.0547, Y 14.7646, Z -5.5000, A 0.000, B 0.000, C 0.000 }
gfCNCPoint4[17300] = {X 407.7575, Y 13.9112, Z -5.5000, A 0.000, B 0.000, C 0.000 }
gfCNCPoint4[17301] = {X 407.6517, Y 13.0137, Z -5.5000, A 0.000, B 0.000, C 0.000 }
gfCNCPoint4[17302] = {X 407.6515, Y 12.1868, Z -5.5000, A 0.000, B 0.000, C 0.000 }
gfCNCPoint4[17303] = {X 407.7558, Y 11.2611, Z -5.5000, A 0.000, B 0.000, C 0.000 }
gfCNCPoint4[17304] = {X 408.0635, Y 10.3819, Z -5.5000, A 0.000, B 0.000, C 0.000 }
gfCNCPoint4[17305] = {X 408.5591, Y 9.5931, Z -5.5000, A 0.000, B 0.000, C 0.000 }
gfCNCPoint4[17306] = {X 409.2178, Y 8.9344, Z -5.5000, A 0.000, B 0.000, C 0.000 }
gfCNCPoint4[17307] = {X 410.0066, Y 8.4388, Z -5.5000, A 0.000, B 0.000, C 0.000 }
gfCNCPoint4[17308] = {X 410.8859, Y 8.1311, Z -5.5000, A 0.000, B 0.000, C 0.000 }
gfCNCPoint4[17309] = {X 411.8115, Y 8.0268, Z -5.5000, A 0.000, B 0.000, C 0.000 }
gfCNCPoint4[17310] = {X 419.3245, Y 8.0268, Z -5.5000, A 0.000, B 0.000, C 0.000 }
gfCNCPoint4[17311] = {X 420.2501, Y 8.1311, Z -5.5000, A 0.000, B 0.000, C 0.000 }
gfCNCPoint4[17312] = {X 421.1294, Y 8.4388, Z -5.5000, A 0.000, B 0.000, C 0.000 }
gfCNCPoint4[17313] = {X 421.9182, Y 8.9344, Z -5.5000, A 0.000, B 0.000, C 0.000 }
gfCNCPoint4[17314] = {X 422.5769, Y 9.5931, Z -5.5000, A 0.000, B 0.000, C 0.000 }
gfCNCPoint4[17315] = {X 423.0725, Y 10.3819, Z -5.5000, A 0.000, B 0.000, C 0.000 }
gfCNCPoint4[17316] = {X 423.3802, Y 11.2611, Z -5.5000, A 0.000, B 0.000, C 0.000 }
gfCNCPoint4[17317] = {X 423.4845, Y 12.1868, Z -5.5000, A 0.000, B 0.000, C 0.000 }
gfCNCPoint4[17318] = {X 423.4845, Y 12.9791, Z -5.5000, A 0.000, B 0.000, C 0.000 }
gfCNCPoint4[17319] = {X 423.3936, Y 13.8210, Z -5.5000, A 0.000, B 0.000, C 0.000 }
gfCNCPoint4[17320] = {X 423.1366, Y 14.6279, Z -5.5000, A 0.000, B 0.000, C 0.000 }
gfCNCPoint4[17321] = {X 422.7238, Y 15.3672, Z -5.5000, A 0.000, B 0.000, C 0.000 }
gfCNCPoint4[17322] = {X 422.1717, Y 16.0093, Z -5.5000, A 0.000, B 0.000, C 0.000 }
gfCNCPoint4[17323] = {X 421.5027, Y 16.5284, Z -5.5000, A 0.000, B 0.000, C 0.000 }
gfCNCPoint4[17324] = {X 420.7435, Y 16.9035, Z -5.5000, A 0.000, B 0.000, C 0.000 }
gfCNCPoint4[17325] = {X 420.0060, Y 17.8914, Z -5.5000, A 0.000, B 0.000, C 0.000 }
gfCNCPoint4[17326] = {X 419.3397, Y 18.9286, Z -5.5000, A 0.000, B 0.000, C 0.000 }
gfCNCPoint4[17327] = {X 417.8582, Y 21.3270, Z -5.5000, A 0.000, B 0.000, C 0.000 }
gfCNCPoint4[17328] = {X 416.0151, Y 24.2871, Z -5.5000, A 0.000, B 0.000, C 0.000 }
gfCNCPoint4[17329] = {X 419.4107, Y 26.4014, Z -5.5000, A 0.000, B 0.000, C 0.000 }
gfCNCPoint4[17330] = {X 415.9472, Y 24.2448, Z -5.5000, A 0.000, B 0.000, C 0.000 }
gfCNCPoint4[17331] = {X 411.3073, Y 31.6966, Z -5.5000, A 0.000, B 0.000, C 0.000 }
gfCNCPoint4[17332] = {X 411.3079, Y 41.0090, Z -5.5000, A 0.000, B 0.000, C 0.000 }
gfCNCPoint4[17333] = {X 411.9448, Y 41.6633, Z -5.5000, A 0.000, B 0.000, C 0.000 }
gfCNCPoint4[17334] = {X 412.4253, Y 42.4398, Z -5.5000, A 0.000, B 0.000, C 0.000 }
gfCNCPoint4[17335] = {X 412.7267, Y 43.3018, Z -5.5000, A 0.000, B 0.000, C 0.000 }
gfCNCPoint4[17336] = {X 412.8347, Y 44.2085, Z -5.5000, A 0.000, B 0.000, C 0.000 }
gfCNCPoint4[17337] = {X 412.8347, Y 45.0002, Z -5.5000, A 0.000, B 0.000, C 0.000 }
gfCNCPoint4[17338] = {X 412.7324, Y 45.9080, Z -5.5000, A 0.000, B 0.000, C 0.000 }
gfCNCPoint4[17339] = {X 412.4306, Y 46.7703, Z -5.5000, A 0.000, B 0.000, C 0.000 }
gfCNCPoint4[17340] = {X 411.9445, Y 47.5439, Z -5.5000, A 0.000, B 0.000, C 0.000 }
gfCNCPoint4[17341] = {X 411.2985, Y 48.1899, Z -5.5000, A 0.000, B 0.000, C 0.000 }
gfCNCPoint4[17342] = {X 410.5249, Y 48.6760, Z -5.5000, A 0.000, B 0.000, C 0.000 }
gfCNCPoint4[17343] = {X 409.6625, Y 48.9777, Z -5.5000, A 0.000, B 0.000, C 0.000 }
gfCNCPoint4[17344] = {X 408.7547, Y 49.0800, Z -5.5000, A 0.000, B 0.000, C 0.000 }
gfCNCPoint4[17345] = {X 402.3112, Y 49.0800, Z -5.5000, A 0.000, B 0.000, C 0.000 }
gfCNCPoint4[17346] = {X 401.4077, Y 48.9787, Z -5.5000, A 0.000, B 0.000, C 0.000 }
gfCNCPoint4[17347] = {X 400.5491, Y 48.6799, Z -5.5000, A 0.000, B 0.000, C 0.000 }
gfCNCPoint4[17348] = {X 399.7780, Y 48.1983, Z -5.5000, A 0.000, B 0.000, C 0.000 }
gfCNCPoint4[17349] = {X 399.1326, Y 47.5579, Z -5.5000, A 0.000, B 0.000, C 0.000 }
gfCNCPoint4[17350] = {X 398.6451, Y 46.7906, Z -5.5000, A 0.000, B 0.000, C 0.000 }
gfCNCPoint4[17351] = {X 398.3396, Y 45.9343, Z -5.5000, A 0.000, B 0.000, C 0.000 }
gfCNCPoint4[17352] = {X 398.2313, Y 45.0316, Z -5.5000, A 0.000, B 0.000, C 0.000 }
gfCNCPoint4[17353] = {X 398.2316, Y 44.1559, Z -5.5000, A 0.000, B 0.000, C 0.000 }
gfCNCPoint4[17354] = {X 398.3416, Y 43.2661, Z -5.5000, A 0.000, B 0.000, C 0.000 }
gfCNCPoint4[17355] = {X 398.6434, Y 42.4218, Z -5.5000, A 0.000, B 0.000, C 0.000 }
gfCNCPoint4[17356] = {X 399.1223, Y 41.6638, Z -5.5000, A 0.000, B 0.000, C 0.000 }
gfCNCPoint4[17357] = {X 399.7552, Y 41.0287, Z -5.5000, A 0.000, B 0.000, C 0.000 }
gfCNCPoint4[17358] = {X 399.7126, Y 31.5364, Z -5.5000, A 0.000, B 0.000, C 0.000 }
gfCNCPoint4[17359] = {X 393.7259, Y 21.1257, Z -5.5000, A 0.000, B 0.000, C 0.000 }
gfCNCPoint4[17360] = {X 392.8355, Y 19.6109, Z -5.5000, A 0.000, B 0.000, C 0.000 }
gfCNCPoint4[17361] = {X 391.9164, Y 18.1134, Z -5.5000, A 0.000, B 0.000, C 0.000 }
gfCNCPoint4[17362] = {X 391.4018, Y 17.4003, Z -5.5000, A 0.000, B 0.000, C 0.000 }
gfCNCPoint4[17363] = {X 390.7989, Y 16.7600, Z -5.5000, A 0.000, B 0.000, C 0.000 }
gfCNCPoint4[17364] = {X 389.9591, Y 16.2987, Z -5.5000, A 0.000, B 0.000, C 0.000 }
gfCNCPoint4[17365] = {X 389.2500, Y 15.6543, Z -5.5000, A 0.000, B 0.000, C 0.000 }
gfCNCPoint4[17366] = {X 388.7108, Y 14.8622, Z -5.5000, A 0.000, B 0.000, C 0.000 }
gfCNCPoint4[17367] = {X 388.3711, Y 13.9663, Z -5.5000, A 0.000, B 0.000, C 0.000 }
gfCNCPoint4[17368] = {X 388.2498, Y 13.0158, Z -5.5000, A 0.000, B 0.000, C 0.000 }
gfCNCPoint4[17369] = {X 388.2496, Y 12.1868, Z -5.5000, A 0.000, B 0.000, C 0.000 }
gfCNCPoint4[17370] = {X 388.3519, Y 11.2789, Z -5.5000, A 0.000, B 0.000, C 0.000 }
gfCNCPoint4[17371] = {X 388.6537, Y 10.4166, Z -5.5000, A 0.000, B 0.000, C 0.000 }
gfCNCPoint4[17372] = {X 389.1398, Y 9.6430, Z -5.5000, A 0.000, B 0.000, C 0.000 }
gfCNCPoint4[17373] = {X 389.7858, Y 8.9969, Z -5.5000, A 0.000, B 0.000, C 0.000 }
gfCNCPoint4[17374] = {X 390.5594, Y 8.5109, Z -5.5000, A 0.000, B 0.000, C 0.000 }
gfCNCPoint4[17375] = {X 391.4217, Y 8.2091, Z -5.5000, A 0.000, B 0.000, C 0.000 }
gfCNCPoint4[17376] = {X 392.3296, Y 8.1068, Z -5.5000, A 0.000, B 0.000, C 0.000 }
gfCNCPoint4[17377] = {X 399.1118, Y 8.1068, Z -5.5000, A 0.000, B 0.000, C 0.000 }
gfCNCPoint4[17378] = {X 400.0196, Y 8.2091, Z -5.5000, A 0.000, B 0.000, C 0.000 }
gfCNCPoint4[17379] = {X 400.8820, Y 8.5109, Z -5.5000, A 0.000, B 0.000, C 0.000 }
gfCNCPoint4[17380] = {X 401.6556, Y 8.9969, Z -5.5000, A 0.000, B 0.000, C 0.000 }
gfCNCPoint4[17381] = {X 402.3016, Y 9.6430, Z -5.5000, A 0.000, B 0.000, C 0.000 }
gfCNCPoint4[17382] = {X 402.7877, Y 10.4166, Z -5.5000, A 0.000, B 0.000, C 0.000 }
gfCNCPoint4[17383] = {X 403.0895, Y 11.2789, Z -5.5000, A 0.000, B 0.000, C 0.000 }
gfCNCPoint4[17384] = {X 403.1918, Y 12.1868, Z -5.5000, A 0.000, B 0.000, C 0.000 }
gfCNCPoint4[17385] = {X 403.1918, Y 12.9782, Z -5.5000, A 0.000, B 0.000, C 0.000 }
gfCNCPoint4[17386] = {X 403.0811, Y 13.9219, Z -5.5000, A 0.000, B 0.000, C 0.000 }
gfCNCPoint4[17387] = {X 402.7551, Y 14.8144, Z -5.5000, A 0.000, B 0.000, C 0.000 }
gfCNCPoint4[17388] = {X 405.3494, Y 19.2899, Z -5.5000, A 0.000, B 0.000, C 0.000 }
gfCNCPoint4[17389] = {X 408.1458, Y 14.7693, Z -5.5000, A 0.000, B 0.000, C 0.000 }
gfCNCPoint4[17390] = {X 408.1091, Y 14.6921, Z -5.5000, A 0.000, B 0.000, C 0.000 }
gfCNCPoint4[17391] = {X 408.0740, Y 14.6141, Z -5.5000, A 0.000, B 0.000, C 0.000 }
gfCNCPoint4[17392] = {X 407.8217, Y 13.8309, Z -5.5000, A 0.000, B 0.000, C 0.000 }
gfCNCPoint4[17393] = {X 407.7317, Y 13.0131, Z -5.5000, A 0.000, B 0.000, C 0.000 }
gfCNCPoint4[17394] = {X 407.7315, Y 12.1868, Z -5.5000, A 0.000, B 0.000, C 0.000 }
gfCNCPoint4[17395] = {X 407.8338, Y 11.2789, Z -5.5000, A 0.000, B 0.000, C 0.000 }
gfCNCPoint4[17396] = {X 408.1356, Y 10.4166, Z -5.5000, A 0.000, B 0.000, C 0.000 }
gfCNCPoint4[17397] = {X 408.6217, Y 9.6430, Z -5.5000, A 0.000, B 0.000, C 0.000 }
gfCNCPoint4[17398] = {X 409.2677, Y 8.9969, Z -5.5000, A 0.000, B 0.000, C 0.000 }
gfCNCPoint4[17399] = {X 410.0413, Y 8.5109, Z -5.5000, A 0.000, B 0.000, C 0.000 }
gfCNCPoint4[17400] = {X 410.9037, Y 8.2091, Z -5.5000, A 0.000, B 0.000, C 0.000 }
gfCNCPoint4[17401] = {X 411.8115, Y 8.1068, Z -5.5000, A 0.000, B 0.000, C 0.000 }
gfCNCPoint4[17402] = {X 419.3245, Y 8.1068, Z -5.5000, A 0.000, B 0.000, C 0.000 }
gfCNCPoint4[17403] = {X 420.2323, Y 8.2091, Z -5.5000, A 0.000, B 0.000, C 0.000 }
gfCNCPoint4[17404] = {X 421.0947, Y 8.5109, Z -5.5000, A 0.000, B 0.000, C 0.000 }
gfCNCPoint4[17405] = {X 421.8683, Y 8.9969, Z -5.5000, A 0.000, B 0.000, C 0.000 }
gfCNCPoint4[17406] = {X 422.5143, Y 9.6430, Z -5.5000, A 0.000, B 0.000, C 0.000 }
gfCNCPoint4[17407] = {X 423.0004, Y 10.4166, Z -5.5000, A 0.000, B 0.000, C 0.000 }
gfCNCPoint4[17408] = {X 423.3022, Y 11.2789, Z -5.5000, A 0.000, B 0.000, C 0.000 }
gfCNCPoint4[17409] = {X 423.4045, Y 12.1868, Z -5.5000, A 0.000, B 0.000, C 0.000 }
gfCNCPoint4[17410] = {X 423.4045, Y 12.9785, Z -5.5000, A 0.000, B 0.000, C 0.000 }
gfCNCPoint4[17411] = {X 423.3146, Y 13.8081, Z -5.5000, A 0.000, B 0.000, C 0.000 }
gfCNCPoint4[17412] = {X 423.0603, Y 14.6027, Z -5.5000, A 0.000, B 0.000, C 0.000 }
gfCNCPoint4[17413] = {X 422.6519, Y 15.3303, Z -5.5000, A 0.000, B 0.000, C 0.000 }
gfCNCPoint4[17414] = {X 422.1061, Y 15.9614, Z -5.5000, A 0.000, B 0.000, C 0.000 }
gfCNCPoint4[17415] = {X 421.4448, Y 16.4702, Z -5.5000, A 0.000, B 0.000, C 0.000 }
gfCNCPoint4[17416] = {X 420.6950, Y 16.8362, Z -5.5000, A 0.000, B 0.000, C 0.000 }
gfCNCPoint4[17417] = {X 419.9468, Y 17.8365, Z -5.5000, A 0.000, B 0.000, C 0.000 }
gfCNCPoint4[17418] = {X 419.2713, Y 18.8871, Z -5.5000, A 0.000, B 0.000, C 0.000 }
gfCNCPoint4[17419] = {X 417.7903, Y 21.2849, Z -5.5000, A 0.000, B 0.000, C 0.000 }
gfCNCPoint4[17420] = {X 415.9472, Y 24.2448, Z -5.5000, A 0.000, B 0.000, C 0.000 }
gfCNCPoint4[17421] = {X 419.3428, Y 26.3591, Z -5.5000, A 0.000, B 0.000, C 0.000 }
gfCNCPoint4[17422] = {X 415.8793, Y 24.2025, Z -5.5000, A 0.000, B 0.000, C 0.000 }
gfCNCPoint4[17423] = {X 411.2273, Y 31.6737, Z -5.5000, A 0.000, B 0.000, C 0.000 }
gfCNCPoint4[17424] = {X 411.2279, Y 41.0470, Z -5.5000, A 0.000, B 0.000, C 0.000 }
gfCNCPoint4[17425] = {X 411.8643, Y 41.6904, Z -5.5000, A 0.000, B 0.000, C 0.000 }
gfCNCPoint4[17426] = {X 412.3449, Y 42.4572, Z -5.5000, A 0.000, B 0.000, C 0.000 }
gfCNCPoint4[17427] = {X 412.6465, Y 43.3104, Z -5.5000, A 0.000, B 0.000, C 0.000 }
gfCNCPoint4[17428] = {X 412.7547, Y 44.2089, Z -5.5000, A 0.000, B 0.000, C 0.000 }
gfCNCPoint4[17429] = {X 412.7545, Y 45.0384, Z -5.5000, A 0.000, B 0.000, C 0.000 }
gfCNCPoint4[17430] = {X 412.6469, Y 45.9222, Z -5.5000, A 0.000, B 0.000, C 0.000 }
gfCNCPoint4[17431] = {X 412.3466, Y 46.7602, Z -5.5000, A 0.000, B 0.000, C 0.000 }
gfCNCPoint4[17432] = {X 411.8683, Y 47.5111, Z -5.5000, A 0.000, B 0.000, C 0.000 }
gfCNCPoint4[17433] = {X 411.2357, Y 48.1376, Z -5.5000, A 0.000, B 0.000, C 0.000 }
gfCNCPoint4[17434] = {X 410.4803, Y 48.6086, Z -5.5000, A 0.000, B 0.000, C 0.000 }
gfCNCPoint4[17435] = {X 409.6394, Y 48.9009, Z -5.5000, A 0.000, B 0.000, C 0.000 }
gfCNCPoint4[17436] = {X 408.7547, Y 49.0000, Z -5.5000, A 0.000, B 0.000, C 0.000 }
gfCNCPoint4[17437] = {X 402.3112, Y 49.0000, Z -5.5000, A 0.000, B 0.000, C 0.000 }
gfCNCPoint4[17438] = {X 401.4211, Y 48.8997, Z -5.5000, A 0.000, B 0.000, C 0.000 }
gfCNCPoint4[17439] = {X 400.5757, Y 48.6039, Z -5.5000, A 0.000, B 0.000, C 0.000 }
gfCNCPoint4[17440] = {X 399.8172, Y 48.1273, Z -5.5000, A 0.000, B 0.000, C 0.000 }
gfCNCPoint4[17441] = {X 399.1839, Y 47.4939, Z -5.5000, A 0.000, B 0.000, C 0.000 }
gfCNCPoint4[17442] = {X 398.7073, Y 46.7355, Z -5.5000, A 0.000, B 0.000, C 0.000 }
gfCNCPoint4[17443] = {X 398.4115, Y 45.8901, Z -5.5000, A 0.000, B 0.000, C 0.000 }
gfCNCPoint4[17444] = {X 398.3112, Y 45.0000, Z -5.5000, A 0.000, B 0.000, C 0.000 }
gfCNCPoint4[17445] = {X 398.3115, Y 44.1569, Z -5.5000, A 0.000, B 0.000, C 0.000 }
gfCNCPoint4[17446] = {X 398.4217, Y 43.2753, Z -5.5000, A 0.000, B 0.000, C 0.000 }
gfCNCPoint4[17447] = {X 398.7237, Y 42.4397, Z -5.5000, A 0.000, B 0.000, C 0.000 }
gfCNCPoint4[17448] = {X 399.2028, Y 41.6913, Z -5.5000, A 0.000, B 0.000, C 0.000 }
gfCNCPoint4[17449] = {X 399.8352, Y 41.0672, Z -5.5000, A 0.000, B 0.000, C 0.000 }
gfCNCPoint4[17450] = {X 399.8370, Y 31.5923, Z -5.5000, A 0.000, B 0.000, C 0.000 }
gfCNCPoint4[17451] = {X 393.7952, Y 21.0858, Z -5.5000, A 0.000, B 0.000, C 0.000 }
gfCNCPoint4[17452] = {X 392.9041, Y 19.5697, Z -5.5000, A 0.000, B 0.000, C 0.000 }
gfCNCPoint4[17453] = {X 391.9842, Y 18.0709, Z -5.5000, A 0.000, B 0.000, C 0.000 }
gfCNCPoint4[17454] = {X 391.4587, Y 17.3436, Z -5.5000, A 0.000, B 0.000, C 0.000 }
gfCNCPoint4[17455] = {X 390.8426, Y 16.6913, Z -5.5000, A 0.000, B 0.000, C 0.000 }
gfCNCPoint4[17456] = {X 390.0091, Y 16.2361, Z -5.5000, A 0.000, B 0.000, C 0.000 }
gfCNCPoint4[17457] = {X 389.3064, Y 15.5972, Z -5.5000, A 0.000, B 0.000, C 0.000 }
gfCNCPoint4[17458] = {X 388.7742, Y 14.8107, Z -5.5000, A 0.000, B 0.000, C 0.000 }
gfCNCPoint4[17459] = {X 388.4423, Y 13.9209, Z -5.5000, A 0.000, B 0.000, C 0.000 }
gfCNCPoint4[17460] = {X 388.3296, Y 12.9779, Z -5.5000, A 0.000, B 0.000, C 0.000 }
gfCNCPoint4[17461] = {X 388.3296, Y 12.1868, Z -5.5000, A 0.000, B 0.000, C 0.000 }
gfCNCPoint4[17462] = {X 388.4299, Y 11.2967, Z -5.5000, A 0.000, B 0.000, C 0.000 }
gfCNCPoint4[17463] = {X 388.7258, Y 10.4513, Z -5.5000, A 0.000, B 0.000, C 0.000 }
gfCNCPoint4[17464] = {X 389.2023, Y 9.6929, Z -5.5000, A 0.000, B 0.000, C 0.000 }
gfCNCPoint4[17465] = {X 389.8357, Y 9.0595, Z -5.5000, A 0.000, B 0.000, C 0.000 }
gfCNCPoint4[17466] = {X 390.5941, Y 8.5829, Z -5.5000, A 0.000, B 0.000, C 0.000 }
gfCNCPoint4[17467] = {X 391.4395, Y 8.2871, Z -5.5000, A 0.000, B 0.000, C 0.000 }
gfCNCPoint4[17468] = {X 392.3296, Y 8.1868, Z -5.5000, A 0.000, B 0.000, C 0.000 }
gfCNCPoint4[17469] = {X 399.1118, Y 8.1868, Z -5.5000, A 0.000, B 0.000, C 0.000 }
gfCNCPoint4[17470] = {X 400.0018, Y 8.2871, Z -5.5000, A 0.000, B 0.000, C 0.000 }
gfCNCPoint4[17471] = {X 400.8473, Y 8.5829, Z -5.5000, A 0.000, B 0.000, C 0.000 }
gfCNCPoint4[17472] = {X 401.6057, Y 9.0595, Z -5.5000, A 0.000, B 0.000, C 0.000 }
gfCNCPoint4[17473] = {X 402.2391, Y 9.6929, Z -5.5000, A 0.000, B 0.000, C 0.000 }
gfCNCPoint4[17474] = {X 402.7156, Y 10.4513, Z -5.5000, A 0.000, B 0.000, C 0.000 }
gfCNCPoint4[17475] = {X 403.0115, Y 11.2967, Z -5.5000, A 0.000, B 0.000, C 0.000 }
gfCNCPoint4[17476] = {X 403.1118, Y 12.1868, Z -5.5000, A 0.000, B 0.000, C 0.000 }
gfCNCPoint4[17477] = {X 403.1115, Y 13.0192, Z -5.5000, A 0.000, B 0.000, C 0.000 }
gfCNCPoint4[17478] = {X 402.9933, Y 13.9442, Z -5.5000, A 0.000, B 0.000, C 0.000 }
gfCNCPoint4[17479] = {X 402.6641, Y 14.8167, Z -5.5000, A 0.000, B 0.000, C 0.000 }
gfCNCPoint4[17480] = {X 405.2576, Y 19.3199, Z -5.5000, A 0.000, B 0.000, C 0.000 }
gfCNCPoint4[17481] = {X 405.3708, Y 19.4076, Z -5.5000, A 0.000, B 0.000, C 0.000 }
gfCNCPoint4[17482] = {X 408.1943, Y 14.8342, Z -5.5000, A 0.000, B 0.000, C 0.000 }
gfCNCPoint4[17483] = {X 408.2428, Y 14.7847, Z -5.5000, A 0.000, B 0.000, C 0.000 }
gfCNCPoint4[17484] = {X 408.1936, Y 14.6840, Z -5.5000, A 0.000, B 0.000, C 0.000 }
gfCNCPoint4[17485] = {X 408.1472, Y 14.5821, Z -5.5000, A 0.000, B 0.000, C 0.000 }
gfCNCPoint4[17486] = {X 407.8964, Y 13.7974, Z -5.5000, A 0.000, B 0.000, C 0.000 }
gfCNCPoint4[17487] = {X 407.8115, Y 12.9780, Z -5.5000, A 0.000, B 0.000, C 0.000 }
gfCNCPoint4[17488] = {X 407.8115, Y 12.1868, Z -5.5000, A 0.000, B 0.000, C 0.000 }
gfCNCPoint4[17489] = {X 407.9118, Y 11.2967, Z -5.5000, A 0.000, B 0.000, C 0.000 }
gfCNCPoint4[17490] = {X 408.2077, Y 10.4513, Z -5.5000, A 0.000, B 0.000, C 0.000 }
gfCNCPoint4[17491] = {X 408.6842, Y 9.6929, Z -5.5000, A 0.000, B 0.000, C 0.000 }
gfCNCPoint4[17492] = {X 409.3176, Y 9.0595, Z -5.5000, A 0.000, B 0.000, C 0.000 }
gfCNCPoint4[17493] = {X 410.0760, Y 8.5829, Z -5.5000, A 0.000, B 0.000, C 0.000 }
gfCNCPoint4[17494] = {X 410.9215, Y 8.2871, Z -5.5000, A 0.000, B 0.000, C 0.000 }
gfCNCPoint4[17495] = {X 411.8115, Y 8.1868, Z -5.5000, A 0.000, B 0.000, C 0.000 }
gfCNCPoint4[17496] = {X 419.3245, Y 8.1868, Z -5.5000, A 0.000, B 0.000, C 0.000 }
gfCNCPoint4[17497] = {X 420.2145, Y 8.2871, Z -5.5000, A 0.000, B 0.000, C 0.000 }
gfCNCPoint4[17498] = {X 421.0600, Y 8.5829, Z -5.5000, A 0.000, B 0.000, C 0.000 }
gfCNCPoint4[17499] = {X 421.8184, Y 9.0595, Z -5.5000, A 0.000, B 0.000, C 0.000 }
gfCNCPoint4[17500] = {X 422.4518, Y 9.6929, Z -5.5000, A 0.000, B 0.000, C 0.000 }
gfCNCPoint4[17501] = {X 422.9283, Y 10.4513, Z -5.5000, A 0.000, B 0.000, C 0.000 }
gfCNCPoint4[17502] = {X 423.2242, Y 11.2967, Z -5.5000, A 0.000, B 0.000, C 0.000 }
gfCNCPoint4[17503] = {X 423.3245, Y 12.1868, Z -5.5000, A 0.000, B 0.000, C 0.000 }
gfCNCPoint4[17504] = {X 423.3245, Y 12.9780, Z -5.5000, A 0.000, B 0.000, C 0.000 }
gfCNCPoint4[17505] = {X 423.1980, Y 13.9554, Z -5.5000, A 0.000, B 0.000, C 0.000 }
gfCNCPoint4[17506] = {X 422.8399, Y 14.8736, Z -5.5000, A 0.000, B 0.000, C 0.000 }
gfCNCPoint4[17507] = {X 422.2713, Y 15.6785, Z -5.5000, A 0.000, B 0.000, C 0.000 }
gfCNCPoint4[17508] = {X 421.5256, Y 16.3229, Z -5.5000, A 0.000, B 0.000, C 0.000 }
gfCNCPoint4[17509] = {X 420.6467, Y 16.7687, Z -5.5000, A 0.000, B 0.000, C 0.000 }
gfCNCPoint4[17510] = {X 419.8876, Y 17.7814, Z -5.5000, A 0.000, B 0.000, C 0.000 }
gfCNCPoint4[17511] = {X 419.2029, Y 18.8457, Z -5.5000, A 0.000, B 0.000, C 0.000 }
gfCNCPoint4[17512] = {X 417.7223, Y 21.2427, Z -5.5000, A 0.000, B 0.000, C 0.000 }
gfCNCPoint4[17513] = {X 415.8793, Y 24.2025, Z -5.5000, A 0.000, B 0.000, C 0.000 }
gfCNCPoint4[17514] = {X 419.3428, Y 26.3591, Z -5.5000, A 0.000, B 0.000, C 0.000 }
gfCNCPoint4[17515] = {X 419.3428, Y 26.3591, Z -2.5000, A 0.000, B 0.000, C 0.000 }
gfCNCPoint4[17516] = {X 419.3428, Y 26.3591, Z 11.0000, A 0.000, B 0.000, C 0.000 }
gfCNCPoint4[17517] = {X 352.3362, Y -3.5323, Z 11.0000, A 0.000, B 0.000, C 0.000 }
gfCNCPoint4[17518] = {X 352.3362, Y -3.5323, Z -2.5000, A 0.000, B 0.000, C 0.000 }
gfCNCPoint4[17519] = {X 352.3362, Y -3.5323, Z -5.5000, A 0.000, B 0.000, C 0.000 }
gfCNCPoint4[17520] = {X 351.5865, Y 0.4782, Z -5.5000, A 0.000, B 0.000, C 0.000 }
gfCNCPoint4[17521] = {X 351.8704, Y 0.5313, Z -5.5000, A 0.000, B 0.000, C 0.000 }
gfCNCPoint4[17522] = {X 353.8209, Y 1.0219, Z -5.5000, A 0.000, B 0.000, C 0.000 }
gfCNCPoint4[17523] = {X 355.7157, Y 1.6966, Z -5.5000, A 0.000, B 0.000, C 0.000 }
gfCNCPoint4[17524] = {X 357.5372, Y 2.5494, Z -5.5000, A 0.000, B 0.000, C 0.000 }
gfCNCPoint4[17525] = {X 359.2689, Y 3.5725, Z -5.5000, A 0.000, B 0.000, C 0.000 }
gfCNCPoint4[17526] = {X 360.8949, Y 4.7564, Z -5.5000, A 0.000, B 0.000, C 0.000 }
gfCNCPoint4[17527] = {X 362.4002, Y 6.0903, Z -5.5000, A 0.000, B 0.000, C 0.000 }
gfCNCPoint4[17528] = {X 363.7712, Y 7.5619, Z -5.5000, A 0.000, B 0.000, C 0.000 }
gfCNCPoint4[17529] = {X 365.1224, Y 9.3183, Z -5.5000, A 0.000, B 0.000, C 0.000 }
gfCNCPoint4[17530] = {X 366.3134, Y 11.1869, Z -5.5000, A 0.000, B 0.000, C 0.000 }
gfCNCPoint4[17531] = {X 367.3349, Y 13.1533, Z -5.5000, A 0.000, B 0.000, C 0.000 }
gfCNCPoint4[17532] = {X 368.1791, Y 15.2022, Z -5.5000, A 0.000, B 0.000, C 0.000 }
gfCNCPoint4[17533] = {X 368.8392, Y 17.3175, Z -5.5000, A 0.000, B 0.000, C 0.000 }
gfCNCPoint4[17534] = {X 369.3103, Y 19.4828, Z -5.5000, A 0.000, B 0.000, C 0.000 }
gfCNCPoint4[17535] = {X 369.6265, Y 21.7093, Z -5.5000, A 0.000, B 0.000, C 0.000 }
gfCNCPoint4[17536] = {X 369.7843, Y 23.9527, Z -5.5000, A 0.000, B 0.000, C 0.000 }
gfCNCPoint4[17537] = {X 369.7828, Y 26.2016, Z -5.5000, A 0.000, B 0.000, C 0.000 }
gfCNCPoint4[17538] = {X 369.6220, Y 28.4447, Z -5.5000, A 0.000, B 0.000, C 0.000 }
gfCNCPoint4[17539] = {X 369.3027, Y 30.6708, Z -5.5000, A 0.000, B 0.000, C 0.000 }
gfCNCPoint4[17540] = {X 368.8017, Y 32.9268, Z -5.5000, A 0.000, B 0.000, C 0.000 }
gfCNCPoint4[17541] = {X 368.0911, Y 35.1258, Z -5.5000, A 0.000, B 0.000, C 0.000 }
gfCNCPoint4[17542] = {X 367.1773, Y 37.2484, Z -5.5000, A 0.000, B 0.000, C 0.000 }
gfCNCPoint4[17543] = {X 366.0681, Y 39.2757, Z -5.5000, A 0.000, B 0.000, C 0.000 }
gfCNCPoint4[17544] = {X 364.7736, Y 41.1900, Z -5.5000, A 0.000, B 0.000, C 0.000 }
gfCNCPoint4[17545] = {X 364.6580, Y 41.3483, Z -5.5000, A 0.000, B 0.000, C 0.000 }
gfCNCPoint4[17546] = {X 363.2576, Y 43.0253, Z -5.5000, A 0.000, B 0.000, C 0.000 }
gfCNCPoint4[17547] = {X 361.6976, Y 44.5550, Z -5.5000, A 0.000, B 0.000, C 0.000 }
gfCNCPoint4[17548] = {X 359.9936, Y 45.9223, Z -5.5000, A 0.000, B 0.000, C 0.000 }
gfCNCPoint4[17549] = {X 358.1622, Y 47.1138, Z -5.5000, A 0.000, B 0.000, C 0.000 }
gfCNCPoint4[17550] = {X 356.2216, Y 48.1175, Z -5.5000, A 0.000, B 0.000, C 0.000 }
gfCNCPoint4[17551] = {X 354.0239, Y 48.9378, Z -5.5000, A 0.000, B 0.000, C 0.000 }
gfCNCPoint4[17552] = {X 351.7542, Y 49.5302, Z -5.5000, A 0.000, B 0.000, C 0.000 }
gfCNCPoint4[17553] = {X 349.4359, Y 49.8886, Z -5.5000, A 0.000, B 0.000, C 0.000 }
gfCNCPoint4[17554] = {X 347.0933, Y 50.0093, Z -5.5000, A 0.000, B 0.000, C 0.000 }
gfCNCPoint4[17555] = {X 345.0267, Y 49.9744, Z -5.5000, A 0.000, B 0.000, C 0.000 }
gfCNCPoint4[17556] = {X 342.9709, Y 49.7604, Z -5.5000, A 0.000, B 0.000, C 0.000 }
gfCNCPoint4[17557] = {X 340.9414, Y 49.3690, Z -5.5000, A 0.000, B 0.000, C 0.000 }
gfCNCPoint4[17558] = {X 338.9536, Y 48.8030, Z -5.5000, A 0.000, B 0.000, C 0.000 }
gfCNCPoint4[17559] = {X 337.0223, Y 48.0667, Z -5.5000, A 0.000, B 0.000, C 0.000 }
gfCNCPoint4[17560] = {X 335.1621, Y 47.1657, Z -5.5000, A 0.000, B 0.000, C 0.000 }
gfCNCPoint4[17561] = {X 333.5778, Y 46.1882, Z -5.5000, A 0.000, B 0.000, C 0.000 }
gfCNCPoint4[17562] = {X 332.0748, Y 45.0897, Z -5.5000, A 0.000, B 0.000, C 0.000 }
gfCNCPoint4[17563] = {X 330.6623, Y 43.8770, Z -5.5000, A 0.000, B 0.000, C 0.000 }
gfCNCPoint4[17564] = {X 329.7213, Y 43.8764, Z -5.5000, A 0.000, B 0.000, C 0.000 }
gfCNCPoint4[17565] = {X 328.8027, Y 43.6721, Z -5.5000, A 0.000, B 0.000, C 0.000 }
gfCNCPoint4[17566] = {X 327.9501, Y 43.2738, Z -5.5000, A 0.000, B 0.000, C 0.000 }
gfCNCPoint4[17567] = {X 327.2040, Y 42.7002, Z -5.5000, A 0.000, B 0.000, C 0.000 }
gfCNCPoint4[17568] = {X 326.5808, Y 42.0925, Z -5.5000, A 0.000, B 0.000, C 0.000 }
gfCNCPoint4[17569] = {X 325.9523, Y 41.3190, Z -5.5000, A 0.000, B 0.000, C 0.000 }
gfCNCPoint4[17570] = {X 325.5179, Y 40.4220, Z -5.5000, A 0.000, B 0.000, C 0.000 }
gfCNCPoint4[17571] = {X 325.3006, Y 39.4493, Z -5.5000, A 0.000, B 0.000, C 0.000 }
gfCNCPoint4[17572] = {X 325.3120, Y 38.4527, Z -5.5000, A 0.000, B 0.000, C 0.000 }
gfCNCPoint4[17573] = {X 325.5514, Y 37.4852, Z -5.5000, A 0.000, B 0.000, C 0.000 }
gfCNCPoint4[17574] = {X 326.0062, Y 36.5984, Z -5.5000, A 0.000, B 0.000, C 0.000 }
gfCNCPoint4[17575] = {X 330.2395, Y 30.2687, Z -5.5000, A 0.000, B 0.000, C 0.000 }
gfCNCPoint4[17576] = {X 330.8409, Y 29.5518, Z -5.5000, A 0.000, B 0.000, C 0.000 }
gfCNCPoint4[17577] = {X 331.5826, Y 28.9812, Z -5.5000, A 0.000, B 0.000, C 0.000 }
gfCNCPoint4[17578] = {X 332.4297, Y 28.5837, Z -5.5000, A 0.000, B 0.000, C 0.000 }
gfCNCPoint4[17579] = {X 333.3425, Y 28.3780, Z -5.5000, A 0.000, B 0.000, C 0.000 }
gfCNCPoint4[17580] = {X 334.2782, Y 28.3736, Z -5.5000, A 0.000, B 0.000, C 0.000 }
gfCNCPoint4[17581] = {X 335.1929, Y 28.5708, Z -5.5000, A 0.000, B 0.000, C 0.000 }
gfCNCPoint4[17582] = {X 336.0437, Y 28.9604, Z -5.5000, A 0.000, B 0.000, C 0.000 }
gfCNCPoint4[17583] = {X 336.7907, Y 29.5240, Z -5.5000, A 0.000, B 0.000, C 0.000 }
gfCNCPoint4[17584] = {X 337.4284, Y 30.1382, Z -5.5000, A 0.000, B 0.000, C 0.000 }
gfCNCPoint4[17585] = {X 337.9528, Y 30.7610, Z -5.5000, A 0.000, B 0.000, C 0.000 }
gfCNCPoint4[17586] = {X 338.3511, Y 31.4711, Z -5.5000, A 0.000, B 0.000, C 0.000 }
gfCNCPoint4[17587] = {X 338.6090, Y 32.2433, Z -5.5000, A 0.000, B 0.000, C 0.000 }
gfCNCPoint4[17588] = {X 338.7175, Y 33.0502, Z -5.5000, A 0.000, B 0.000, C 0.000 }
gfCNCPoint4[17589] = {X 338.6726, Y 33.8631, Z -5.5000, A 0.000, B 0.000, C 0.000 }
gfCNCPoint4[17590] = {X 339.4392, Y 34.5528, Z -5.5000, A 0.000, B 0.000, C 0.000 }
gfCNCPoint4[17591] = {X 340.2350, Y 35.2087, Z -5.5000, A 0.000, B 0.000, C 0.000 }
gfCNCPoint4[17592] = {X 341.5323, Y 36.0601, Z -5.5000, A 0.000, B 0.000, C 0.000 }
gfCNCPoint4[17593] = {X 342.9398, Y 36.7134, Z -5.5000, A 0.000, B 0.000, C 0.000 }
gfCNCPoint4[17594] = {X 344.4275, Y 37.1546, Z -5.5000, A 0.000, B 0.000, C 0.000 }
gfCNCPoint4[17595] = {X 345.9637, Y 37.3743, Z -5.5000, A 0.000, B 0.000, C 0.000 }
gfCNCPoint4[17596] = {X 347.5154, Y 37.3679, Z -5.5000, A 0.000, B 0.000, C 0.000 }
gfCNCPoint4[17597] = {X 348.9563, Y 37.1749, Z -5.5000, A 0.000, B 0.000, C 0.000 }
gfCNCPoint4[17598] = {X 350.3465, Y 36.7497, Z -5.5000, A 0.000, B 0.000, C 0.000 }
gfCNCPoint4[17599] = {X 351.6489, Y 36.1038, Z -5.5000, A 0.000, B 0.000, C 0.000 }
gfCNCPoint4[17600] = {X 352.8287, Y 35.2543, Z -5.5000, A 0.000, B 0.000, C 0.000 }
gfCNCPoint4[17601] = {X 353.9823, Y 34.1335, Z -5.5000, A 0.000, B 0.000, C 0.000 }
gfCNCPoint4[17602] = {X 354.9806, Y 32.8725, Z -5.5000, A 0.000, B 0.000, C 0.000 }
gfCNCPoint4[17603] = {X 355.8068, Y 31.4926, Z -5.5000, A 0.000, B 0.000, C 0.000 }
gfCNCPoint4[17604] = {X 356.4468, Y 30.0171, Z -5.5000, A 0.000, B 0.000, C 0.000 }
gfCNCPoint4[17605] = {X 356.8898, Y 28.4710, Z -5.5000, A 0.000, B 0.000, C 0.000 }
gfCNCPoint4[17606] = {X 357.1631, Y 26.7828, Z -5.5000, A 0.000, B 0.000, C 0.000 }
gfCNCPoint4[17607] = {X 357.2744, Y 25.0762, Z -5.5000, A 0.000, B 0.000, C 0.000 }
gfCNCPoint4[17608] = {X 357.2227, Y 23.3668, Z -5.5000, A 0.000, B 0.000, C 0.000 }
gfCNCPoint4[17609] = {X 357.0085, Y 21.6701, Z -5.5000, A 0.000, B 0.000, C 0.000 }
gfCNCPoint4[17610] = {X 356.6547, Y 20.1541, Z -5.5000, A 0.000, B 0.000, C 0.000 }
gfCNCPoint4[17611] = {X 356.1051, Y 18.6977, Z -5.5000, A 0.000, B 0.000, C 0.000 }
gfCNCPoint4[17612] = {X 355.3690, Y 17.3259, Z -5.5000, A 0.000, B 0.000, C 0.000 }
gfCNCPoint4[17613] = {X 354.4594, Y 16.0626, Z -5.5000, A 0.000, B 0.000, C 0.000 }
gfCNCPoint4[17614] = {X 353.5887, Y 15.1357, Z -5.5000, A 0.000, B 0.000, C 0.000 }
gfCNCPoint4[17615] = {X 352.5980, Y 14.3384, Z -5.5000, A 0.000, B 0.000, C 0.000 }
gfCNCPoint4[17616] = {X 351.5062, Y 13.6862, Z -5.5000, A 0.000, B 0.000, C 0.000 }
gfCNCPoint4[17617] = {X 350.3346, Y 13.1917, Z -5.5000, A 0.000, B 0.000, C 0.000 }
gfCNCPoint4[17618] = {X 349.1057, Y 12.8644, Z -5.5000, A 0.000, B 0.000, C 0.000 }
gfCNCPoint4[17619] = {X 347.3454, Y 12.6454, Z -5.5000, A 0.000, B 0.000, C 0.000 }
gfCNCPoint4[17620] = {X 345.5715, Y 12.6612, Z -5.5000, A 0.000, B 0.000, C 0.000 }
gfCNCPoint4[17621] = {X 343.8154, Y 12.9115, Z -5.5000, A 0.000, B 0.000, C 0.000 }
gfCNCPoint4[17622] = {X 342.1077, Y 13.3919, Z -5.5000, A 0.000, B 0.000, C 0.000 }
gfCNCPoint4[17623] = {X 340.4787, Y 14.0939, Z -5.5000, A 0.000, B 0.000, C 0.000 }
gfCNCPoint4[17624] = {X 338.9568, Y 15.0053, Z -5.5000, A 0.000, B 0.000, C 0.000 }
gfCNCPoint4[17625] = {X 338.9179, Y 15.8500, Z -5.5000, A 0.000, B 0.000, C 0.000 }
gfCNCPoint4[17626] = {X 338.7152, Y 16.6710, Z -5.5000, A 0.000, B 0.000, C 0.000 }
gfCNCPoint4[17627] = {X 338.3564, Y 17.4367, Z -5.5000, A 0.000, B 0.000, C 0.000 }
gfCNCPoint4[17628] = {X 337.8553, Y 18.1179, Z -5.5000, A 0.000, B 0.000, C 0.000 }
gfCNCPoint4[17629] = {X 337.2312, Y 18.6885, Z -5.5000, A 0.000, B 0.000, C 0.000 }
gfCNCPoint4[17630] = {X 336.5140, Y 19.2162, Z -5.5000, A 0.000, B 0.000, C 0.000 }
gfCNCPoint4[17631] = {X 335.6982, Y 19.6754, Z -5.5000, A 0.000, B 0.000, C 0.000 }
gfCNCPoint4[17632] = {X 334.8027, Y 19.9480, Z -5.5000, A 0.000, B 0.000, C 0.000 }
gfCNCPoint4[17633] = {X 333.8694, Y 20.0213, Z -5.5000, A 0.000, B 0.000, C 0.000 }
gfCNCPoint4[17634] = {X 332.9422, Y 19.8919, Z -5.5000, A 0.000, B 0.000, C 0.000 }
gfCNCPoint4[17635] = {X 332.0647, Y 19.5657, Z -5.5000, A 0.000, B 0.000, C 0.000 }
gfCNCPoint4[17636] = {X 331.2781, Y 19.0581, Z -5.5000, A 0.000, B 0.000, C 0.000 }
gfCNCPoint4[17637] = {X 330.6193, Y 18.3931, Z -5.5000, A 0.000, B 0.000, C 0.000 }
gfCNCPoint4[17638] = {X 330.1192, Y 17.6017, Z -5.5000, A 0.000, B 0.000, C 0.000 }
gfCNCPoint4[17639] = {X 326.5942, Y 10.3502, Z -5.5000, A 0.000, B 0.000, C 0.000 }
gfCNCPoint4[17640] = {X 326.2930, Y 9.5271, Z -5.5000, A 0.000, B 0.000, C 0.000 }
gfCNCPoint4[17641] = {X 326.1640, Y 8.6602, Z -5.5000, A 0.000, B 0.000, C 0.000 }
gfCNCPoint4[17642] = {X 326.2128, Y 7.7851, Z -5.5000, A 0.000, B 0.000, C 0.000 }
gfCNCPoint4[17643] = {X 326.4371, Y 6.9378, Z -5.5000, A 0.000, B 0.000, C 0.000 }
gfCNCPoint4[17644] = {X 326.8279, Y 6.1532, Z -5.5000, A 0.000, B 0.000, C 0.000 }
gfCNCPoint4[17645] = {X 327.3690, Y 5.4637, Z -5.5000, A 0.000, B 0.000, C 0.000 }
gfCNCPoint4[17646] = {X 328.0381, Y 4.8976, Z -5.5000, A 0.000, B 0.000, C 0.000 }
gfCNCPoint4[17647] = {X 328.7084, Y 4.4386, Z -5.5000, A 0.000, B 0.000, C 0.000 }
gfCNCPoint4[17648] = {X 329.5888, Y 3.9824, Z -5.5000, A 0.000, B 0.000, C 0.000 }
gfCNCPoint4[17649] = {X 330.5500, Y 3.7391, Z -5.5000, A 0.000, B 0.000, C 0.000 }
gfCNCPoint4[17650] = {X 331.5413, Y 3.7213, Z -5.5000, A 0.000, B 0.000, C 0.000 }
gfCNCPoint4[17651] = {X 332.5106, Y 3.9300, Z -5.5000, A 0.000, B 0.000, C 0.000 }
gfCNCPoint4[17652] = {X 333.9975, Y 3.1003, Z -5.5000, A 0.000, B 0.000, C 0.000 }
gfCNCPoint4[17653] = {X 335.5315, Y 2.3613, Z -5.5000, A 0.000, B 0.000, C 0.000 }
gfCNCPoint4[17654] = {X 337.6677, Y 1.4947, Z -5.5000, A 0.000, B 0.000, C 0.000 }
gfCNCPoint4[17655] = {X 339.8716, Y 0.8186, Z -5.5000, A 0.000, B 0.000, C 0.000 }
gfCNCPoint4[17656] = {X 342.1263, Y 0.3383, Z -5.5000, A 0.000, B 0.000, C 0.000 }
gfCNCPoint4[17657] = {X 344.4144, Y 0.0574, Z -5.5000, A 0.000, B 0.000, C 0.000 }
gfCNCPoint4[17658] = {X 346.7183, Y -0.0219, Z -5.5000, A 0.000, B 0.000, C 0.000 }
gfCNCPoint4[17659] = {X 349.0203, Y 0.1010, Z -5.5000, A 0.000, B 0.000, C 0.000 }
gfCNCPoint4[17660] = {X 351.3026, Y 0.4252, Z -5.5000, A 0.000, B 0.000, C 0.000 }
gfCNCPoint4[17661] = {X 351.5865, Y 0.4782, Z -5.5000, A 0.000, B 0.000, C 0.000 }
gfCNCPoint4[17662] = {X 352.3215, Y -3.4537, Z -5.5000, A 0.000, B 0.000, C 0.000 }
gfCNCPoint4[17663] = {X 351.5718, Y 0.5569, Z -5.5000, A 0.000, B 0.000, C 0.000 }
gfCNCPoint4[17664] = {X 351.8551, Y 0.6098, Z -5.5000, A 0.000, B 0.000, C 0.000 }
gfCNCPoint4[17665] = {X 353.7982, Y 1.0986, Z -5.5000, A 0.000, B 0.000, C 0.000 }
gfCNCPoint4[17666] = {X 355.6856, Y 1.7708, Z -5.5000, A 0.000, B 0.000, C 0.000 }
gfCNCPoint4[17667] = {X 357.5002, Y 2.6203, Z -5.5000, A 0.000, B 0.000, C 0.000 }
gfCNCPoint4[17668] = {X 359.2252, Y 3.6395, Z -5.5000, A 0.000, B 0.000, C 0.000 }
gfCNCPoint4[17669] = {X 360.8449, Y 4.8188, Z -5.5000, A 0.000, B 0.000, C 0.000 }
gfCNCPoint4[17670] = {X 362.3444, Y 6.1476, Z -5.5000, A 0.000, B 0.000, C 0.000 }
gfCNCPoint4[17671] = {X 363.7101, Y 7.6136, Z -5.5000, A 0.000, B 0.000, C 0.000 }
gfCNCPoint4[17672] = {X 365.0570, Y 9.3644, Z -5.5000, A 0.000, B 0.000, C 0.000 }
gfCNCPoint4[17673] = {X 366.2442, Y 11.2271, Z -5.5000, A 0.000, B 0.000, C 0.000 }
gfCNCPoint4[17674] = {X 367.2625, Y 13.1872, Z -5.5000, A 0.000, B 0.000, C 0.000 }
gfCNCPoint4[17675] = {X 368.1039, Y 15.2296, Z -5.5000, A 0.000, B 0.000, C 0.000 }
gfCNCPoint4[17676] = {X 368.7620, Y 17.3381, Z -5.5000, A 0.000, B 0.000, C 0.000 }
gfCNCPoint4[17677] = {X 369.2315, Y 19.4965, Z -5.5000, A 0.000, B 0.000, C 0.000 }
gfCNCPoint4[17678] = {X 369.5470, Y 21.7176, Z -5.5000, A 0.000, B 0.000, C 0.000 }
gfCNCPoint4[17679] = {X 369.7044, Y 23.9554, Z -5.5000, A 0.000, B 0.000, C 0.000 }
gfCNCPoint4[17680] = {X 369.7029, Y 26.1987, Z -5.5000, A 0.000, B 0.000, C 0.000 }
gfCNCPoint4[17681] = {X 369.5424, Y 28.4363, Z -5.5000, A 0.000, B 0.000, C 0.000 }
gfCNCPoint4[17682] = {X 369.2240, Y 30.6569, Z -5.5000, A 0.000, B 0.000, C 0.000 }
gfCNCPoint4[17683] = {X 368.7246, Y 32.9057, Z -5.5000, A 0.000, B 0.000, C 0.000 }
gfCNCPoint4[17684] = {X 368.0163, Y 35.0976, Z -5.5000, A 0.000, B 0.000, C 0.000 }
gfCNCPoint4[17685] = {X 367.1053, Y 37.2134, Z -5.5000, A 0.000, B 0.000, C 0.000 }
gfCNCPoint4[17686] = {X 365.9997, Y 39.2343, Z -5.5000, A 0.000, B 0.000, C 0.000 }
gfCNCPoint4[17687] = {X 364.7092, Y 41.1425, Z -5.5000, A 0.000, B 0.000, C 0.000 }
gfCNCPoint4[17688] = {X 364.5937, Y 41.3007, Z -5.5000, A 0.000, B 0.000, C 0.000 }
gfCNCPoint4[17689] = {X 363.1986, Y 42.9713, Z -5.5000, A 0.000, B 0.000, C 0.000 }
gfCNCPoint4[17690] = {X 361.6445, Y 44.4952, Z -5.5000, A 0.000, B 0.000, C 0.000 }
gfCNCPoint4[17691] = {X 359.9468, Y 45.8574, Z -5.5000, A 0.000, B 0.000, C 0.000 }
gfCNCPoint4[17692] = {X 358.1224, Y 47.0444, Z -5.5000, A 0.000, B 0.000, C 0.000 }
gfCNCPoint4[17693] = {X 356.1891, Y 48.0444, Z -5.5000, A 0.000, B 0.000, C 0.000 }
gfCNCPoint4[17694] = {X 353.9990, Y 48.8618, Z -5.5000, A 0.000, B 0.000, C 0.000 }
gfCNCPoint4[17695] = {X 351.7371, Y 49.4520, Z -5.5000, A 0.000, B 0.000, C 0.000 }
gfCNCPoint4[17696] = {X 349.4268, Y 49.8091, Z -5.5000, A 0.000, B 0.000, C 0.000 }
gfCNCPoint4[17697] = {X 347.0922, Y 49.9293, Z -5.5000, A 0.000, B 0.000, C 0.000 }
gfCNCPoint4[17698] = {X 345.0325, Y 49.8946, Z -5.5000, A 0.000, B 0.000, C 0.000 }
gfCNCPoint4[17699] = {X 342.9836, Y 49.6814, Z -5.5000, A 0.000, B 0.000, C 0.000 }
gfCNCPoint4[17700] = {X 340.9609, Y 49.2914, Z -5.5000, A 0.000, B 0.000, C 0.000 }
gfCNCPoint4[17701] = {X 338.9796, Y 48.7273, Z -5.5000, A 0.000, B 0.000, C 0.000 }
gfCNCPoint4[17702] = {X 337.0547, Y 47.9936, Z -5.5000, A 0.000, B 0.000, C 0.000 }
gfCNCPoint4[17703] = {X 335.2008, Y 47.0957, Z -5.5000, A 0.000, B 0.000, C 0.000 }
gfCNCPoint4[17704] = {X 333.6118, Y 46.1147, Z -5.5000, A 0.000, B 0.000, C 0.000 }
gfCNCPoint4[17705] = {X 332.1051, Y 45.0117, Z -5.5000, A 0.000, B 0.000, C 0.000 }
gfCNCPoint4[17706] = {X 330.6899, Y 43.7934, Z -5.5000, A 0.000, B 0.000, C 0.000 }
gfCNCPoint4[17707] = {X 329.7572, Y 43.7998, Z -5.5000, A 0.000, B 0.000, C 0.000 }
gfCNCPoint4[17708] = {X 328.8457, Y 43.6022, Z -5.5000, A 0.000, B 0.000, C 0.000 }
gfCNCPoint4[17709] = {X 327.9994, Y 43.2101, Z -5.5000, A 0.000, B 0.000, C 0.000 }
gfCNCPoint4[17710] = {X 327.2594, Y 42.6425, Z -5.5000, A 0.000, B 0.000, C 0.000 }
gfCNCPoint4[17711] = {X 326.6366, Y 42.0352, Z -5.5000, A 0.000, B 0.000, C 0.000 }
gfCNCPoint4[17712] = {X 326.0198, Y 41.2760, Z -5.5000, A 0.000, B 0.000, C 0.000 }
gfCNCPoint4[17713] = {X 325.5934, Y 40.3956, Z -5.5000, A 0.000, B 0.000, C 0.000 }
gfCNCPoint4[17714] = {X 325.3802, Y 39.4410, Z -5.5000, A 0.000, B 0.000, C 0.000 }
gfCNCPoint4[17715] = {X 325.3913, Y 38.4628, Z -5.5000, A 0.000, B 0.000, C 0.000 }
gfCNCPoint4[17716] = {X 325.6264, Y 37.5133, Z -5.5000, A 0.000, B 0.000, C 0.000 }
gfCNCPoint4[17717] = {X 326.0727, Y 36.6429, Z -5.5000, A 0.000, B 0.000, C 0.000 }
gfCNCPoint4[17718] = {X 330.3060, Y 30.3132, Z -5.5000, A 0.000, B 0.000, C 0.000 }
gfCNCPoint4[17719] = {X 330.8963, Y 29.6095, Z -5.5000, A 0.000, B 0.000, C 0.000 }
gfCNCPoint4[17720] = {X 331.6242, Y 29.0495, Z -5.5000, A 0.000, B 0.000, C 0.000 }
gfCNCPoint4[17721] = {X 332.4556, Y 28.6594, Z -5.5000, A 0.000, B 0.000, C 0.000 }
gfCNCPoint4[17722] = {X 333.3515, Y 28.4575, Z -5.5000, A 0.000, B 0.000, C 0.000 }
gfCNCPoint4[17723] = {X 334.2699, Y 28.4532, Z -5.5000, A 0.000, B 0.000, C 0.000 }
gfCNCPoint4[17724] = {X 335.1677, Y 28.6467, Z -5.5000, A 0.000, B 0.000, C 0.000 }
gfCNCPoint4[17725] = {X 336.0027, Y 29.0291, Z -5.5000, A 0.000, B 0.000, C 0.000 }
gfCNCPoint4[17726] = {X 336.7358, Y 29.5823, Z -5.5000, A 0.000, B 0.000, C 0.000 }
gfCNCPoint4[17727] = {X 337.3723, Y 30.1953, Z -5.5000, A 0.000, B 0.000, C 0.000 }
gfCNCPoint4[17728] = {X 337.8918, Y 30.8134, Z -5.5000, A 0.000, B 0.000, C 0.000 }
gfCNCPoint4[17729] = {X 338.2846, Y 31.5188, Z -5.5000, A 0.000, B 0.000, C 0.000 }
gfCNCPoint4[17730] = {X 338.5367, Y 32.2858, Z -5.5000, A 0.000, B 0.000, C 0.000 }
gfCNCPoint4[17731] = {X 338.6387, Y 33.0867, Z -5.5000, A 0.000, B 0.000, C 0.000 }
gfCNCPoint4[17732] = {X 338.5871, Y 33.8925, Z -5.5000, A 0.000, B 0.000, C 0.000 }
gfCNCPoint4[17733] = {X 339.3712, Y 34.5998, Z -5.5000, A 0.000, B 0.000, C 0.000 }
gfCNCPoint4[17734] = {X 340.1859, Y 35.2718, Z -5.5000, A 0.000, B 0.000, C 0.000 }
gfCNCPoint4[17735] = {X 341.4928, Y 36.1297, Z -5.5000, A 0.000, B 0.000, C 0.000 }
gfCNCPoint4[17736] = {X 342.9108, Y 36.7879, Z -5.5000, A 0.000, B 0.000, C 0.000 }
gfCNCPoint4[17737] = {X 344.4096, Y 37.2326, Z -5.5000, A 0.000, B 0.000, C 0.000 }
gfCNCPoint4[17738] = {X 345.9572, Y 37.4541, Z -5.5000, A 0.000, B 0.000, C 0.000 }
gfCNCPoint4[17739] = {X 347.5205, Y 37.4478, Z -5.5000, A 0.000, B 0.000, C 0.000 }
gfCNCPoint4[17740] = {X 348.6863, Y 37.3109, Z -5.5000, A 0.000, B 0.000, C 0.000 }
gfCNCPoint4[17741] = {X 349.8242, Y 37.0230, Z -5.5000, A 0.000, B 0.000, C 0.000 }
gfCNCPoint4[17742] = {X 350.9148, Y 36.5891, Z -5.5000, A 0.000, B 0.000, C 0.000 }
gfCNCPoint4[17743] = {X 351.9394, Y 36.0165, Z -5.5000, A 0.000, B 0.000, C 0.000 }
gfCNCPoint4[17744] = {X 352.8806, Y 35.3152, Z -5.5000, A 0.000, B 0.000, C 0.000 }
gfCNCPoint4[17745] = {X 354.0417, Y 34.1872, Z -5.5000, A 0.000, B 0.000, C 0.000 }
gfCNCPoint4[17746] = {X 355.0465, Y 32.9180, Z -5.5000, A 0.000, B 0.000, C 0.000 }
gfCNCPoint4[17747] = {X 355.8780, Y 31.5291, Z -5.5000, A 0.000, B 0.000, C 0.000 }
gfCNCPoint4[17748] = {X 356.5221, Y 30.0440, Z -5.5000, A 0.000, B 0.000, C 0.000 }
gfCNCPoint4[17749] = {X 356.9680, Y 28.4878, Z -5.5000, A 0.000, B 0.000, C 0.000 }
gfCNCPoint4[17750] = {X 357.2425, Y 26.7920, Z -5.5000, A 0.000, B 0.000, C 0.000 }
gfCNCPoint4[17751] = {X 357.3544, Y 25.0778, Z -5.5000, A 0.000, B 0.000, C 0.000 }
gfCNCPoint4[17752] = {X 357.3025, Y 23.3607, Z -5.5000, A 0.000, B 0.000, C 0.000 }
gfCNCPoint4[17753] = {X 357.0873, Y 21.6563, Z -5.5000, A 0.000, B 0.000, C 0.000 }
gfCNCPoint4[17754] = {X 356.7311, Y 20.1303, Z -5.5000, A 0.000, B 0.000, C 0.000 }
gfCNCPoint4[17755] = {X 356.1777, Y 18.6642, Z -5.5000, A 0.000, B 0.000, C 0.000 }
gfCNCPoint4[17756] = {X 355.4368, Y 17.2834, Z -5.5000, A 0.000, B 0.000, C 0.000 }
gfCNCPoint4[17757] = {X 354.5211, Y 16.0117, Z -5.5000, A 0.000, B 0.000, C 0.000 }
gfCNCPoint4[17758] = {X 353.6429, Y 15.0768, Z -5.5000, A 0.000, B 0.000, C 0.000 }
gfCNCPoint4[17759] = {X 352.6435, Y 14.2726, Z -5.5000, A 0.000, B 0.000, C 0.000 }
gfCNCPoint4[17760] = {X 351.5422, Y 13.6148, Z -5.5000, A 0.000, B 0.000, C 0.000 }
gfCNCPoint4[17761] = {X 350.3604, Y 13.1160, Z -5.5000, A 0.000, B 0.000, C 0.000 }
gfCNCPoint4[17762] = {X 349.1209, Y 12.7858, Z -5.5000, A 0.000, B 0.000, C 0.000 }
gfCNCPoint4[17763] = {X 347.3425, Y 12.5651, Z -5.5000, A 0.000, B 0.000, C 0.000 }
gfCNCPoint4[17764] = {X 345.5506, Y 12.5826, Z -5.5000, A 0.000, B 0.000, C 0.000 }
gfCNCPoint4[17765] = {X 343.7769, Y 12.8379, Z -5.5000, A 0.000, B 0.000, C 0.000 }
gfCNCPoint4[17766] = {X 342.0528, Y 13.3265, Z -5.5000, A 0.000, B 0.000, C 0.000 }
gfCNCPoint4[17767] = {X 340.4089, Y 14.0398, Z -5.5000, A 0.000, B 0.000, C 0.000 }
gfCNCPoint4[17768] = {X 338.8744, Y 14.9652, Z -5.5000, A 0.000, B 0.000, C 0.000 }
gfCNCPoint4[17769] = {X 338.8437, Y 15.8034, Z -5.5000, A 0.000, B 0.000, C 0.000 }
gfCNCPoint4[17770] = {X 338.6485, Y 16.6192, Z -5.5000, A 0.000, B 0.000, C 0.000 }
gfCNCPoint4[17771] = {X 338.2967, Y 17.3806, Z -5.5000, A 0.000, B 0.000, C 0.000 }
gfCNCPoint4[17772] = {X 337.8018, Y 18.0578, Z -5.5000, A 0.000, B 0.000, C 0.000 }
gfCNCPoint4[17773] = {X 337.1832, Y 18.6244, Z -5.5000, A 0.000, B 0.000, C 0.000 }
gfCNCPoint4[17774] = {X 336.4675, Y 19.1512, Z -5.5000, A 0.000, B 0.000, C 0.000 }
gfCNCPoint4[17775] = {X 335.6668, Y 19.6018, Z -5.5000, A 0.000, B 0.000, C 0.000 }
gfCNCPoint4[17776] = {X 334.7878, Y 19.8694, Z -5.5000, A 0.000, B 0.000, C 0.000 }
gfCNCPoint4[17777] = {X 333.8718, Y 19.9414, Z -5.5000, A 0.000, B 0.000, C 0.000 }
gfCNCPoint4[17778] = {X 332.9618, Y 19.8143, Z -5.5000, A 0.000, B 0.000, C 0.000 }
gfCNCPoint4[17779] = {X 332.1006, Y 19.4942, Z -5.5000, A 0.000, B 0.000, C 0.000 }
gfCNCPoint4[17780] = {X 331.3285, Y 18.9960, Z -5.5000, A 0.000, B 0.000, C 0.000 }
gfCNCPoint4[17781] = {X 330.6819, Y 18.3433, Z -5.5000, A 0.000, B 0.000, C 0.000 }
gfCNCPoint4[17782] = {X 330.1911, Y 17.5665, Z -5.5000, A 0.000, B 0.000, C 0.000 }
gfCNCPoint4[17783] = {X 326.6662, Y 10.3152, Z -5.5000, A 0.000, B 0.000, C 0.000 }
gfCNCPoint4[17784] = {X 326.3374, Y 9.3676, Z -5.5000, A 0.000, B 0.000, C 0.000 }
gfCNCPoint4[17785] = {X 326.2405, Y 8.3693, Z -5.5000, A 0.000, B 0.000, C 0.000 }
gfCNCPoint4[17786] = {X 326.3807, Y 7.3762, Z -5.5000, A 0.000, B 0.000, C 0.000 }
gfCNCPoint4[17787] = {X 326.7504, Y 6.4438, Z -5.5000, A 0.000, B 0.000, C 0.000 }
gfCNCPoint4[17788] = {X 327.3287, Y 5.6243, Z -5.5000, A 0.000, B 0.000, C 0.000 }
gfCNCPoint4[17789] = {X 328.0833, Y 4.9636, Z -5.5000, A 0.000, B 0.000, C 0.000 }
gfCNCPoint4[17790] = {X 328.7533, Y 4.5047, Z -5.5000, A 0.000, B 0.000, C 0.000 }
gfCNCPoint4[17791] = {X 329.6260, Y 4.0539, Z -5.5000, A 0.000, B 0.000, C 0.000 }
gfCNCPoint4[17792] = {X 330.5790, Y 3.8160, Z -5.5000, A 0.000, B 0.000, C 0.000 }
gfCNCPoint4[17793] = {X 331.5612, Y 3.8037, Z -5.5000, A 0.000, B 0.000, C 0.000 }
gfCNCPoint4[17794] = {X 332.5198, Y 4.0178, Z -5.5000, A 0.000, B 0.000, C 0.000 }
gfCNCPoint4[17795] = {X 334.0181, Y 3.1797, Z -5.5000, A 0.000, B 0.000, C 0.000 }
gfCNCPoint4[17796] = {X 335.5644, Y 2.4342, Z -5.5000, A 0.000, B 0.000, C 0.000 }
gfCNCPoint4[17797] = {X 337.6942, Y 1.5702, Z -5.5000, A 0.000, B 0.000, C 0.000 }
gfCNCPoint4[17798] = {X 339.8914, Y 0.8961, Z -5.5000, A 0.000, B 0.000, C 0.000 }
gfCNCPoint4[17799] = {X 342.1393, Y 0.4172, Z -5.5000, A 0.000, B 0.000, C 0.000 }
gfCNCPoint4[17800] = {X 344.4205, Y 0.1372, Z -5.5000, A 0.000, B 0.000, C 0.000 }
gfCNCPoint4[17801] = {X 346.7174, Y 0.0581, Z -5.5000, A 0.000, B 0.000, C 0.000 }
gfCNCPoint4[17802] = {X 349.0124, Y 0.1806, Z -5.5000, A 0.000, B 0.000, C 0.000 }
gfCNCPoint4[17803] = {X 351.2879, Y 0.5038, Z -5.5000, A 0.000, B 0.000, C 0.000 }
gfCNCPoint4[17804] = {X 351.5718, Y 0.5569, Z -5.5000, A 0.000, B 0.000, C 0.000 }
gfCNCPoint4[17805] = {X 352.3068, Y -3.3750, Z -5.5000, A 0.000, B 0.000, C 0.000 }
gfCNCPoint4[17806] = {X 351.5571, Y 0.6355, Z -5.5000, A 0.000, B 0.000, C 0.000 }
gfCNCPoint4[17807] = {X 351.8399, Y 0.6884, Z -5.5000, A 0.000, B 0.000, C 0.000 }
gfCNCPoint4[17808] = {X 353.7754, Y 1.1752, Z -5.5000, A 0.000, B 0.000, C 0.000 }
gfCNCPoint4[17809] = {X 355.6556, Y 1.8449, Z -5.5000, A 0.000, B 0.000, C 0.000 }
gfCNCPoint4[17810] = {X 357.4631, Y 2.6912, Z -5.5000, A 0.000, B 0.000, C 0.000 }
gfCNCPoint4[17811] = {X 359.1814, Y 3.7064, Z -5.5000, A 0.000, B 0.000, C 0.000 }
gfCNCPoint4[17812] = {X 360.7949, Y 4.8813, Z -5.5000, A 0.000, B 0.000, C 0.000 }
gfCNCPoint4[17813] = {X 362.2886, Y 6.2049, Z -5.5000, A 0.000, B 0.000, C 0.000 }
gfCNCPoint4[17814] = {X 363.6490, Y 7.6653, Z -5.5000, A 0.000, B 0.000, C 0.000 }
gfCNCPoint4[17815] = {X 364.9916, Y 9.4104, Z -5.5000, A 0.000, B 0.000, C 0.000 }
gfCNCPoint4[17816] = {X 366.1750, Y 11.2672, Z -5.5000, A 0.000, B 0.000, C 0.000 }
gfCNCPoint4[17817] = {X 367.1900, Y 13.2211, Z -5.5000, A 0.000, B 0.000, C 0.000 }
gfCNCPoint4[17818] = {X 368.0288, Y 15.2570, Z -5.5000, A 0.000, B 0.000, C 0.000 }
gfCNCPoint4[17819] = {X 368.6847, Y 17.3588, Z -5.5000, A 0.000, B 0.000, C 0.000 }
gfCNCPoint4[17820] = {X 369.1527, Y 19.5104, Z -5.5000, A 0.000, B 0.000, C 0.000 }
gfCNCPoint4[17821] = {X 369.4674, Y 21.7259, Z -5.5000, A 0.000, B 0.000, C 0.000 }
gfCNCPoint4[17822] = {X 369.6244, Y 23.9581, Z -5.5000, A 0.000, B 0.000, C 0.000 }
gfCNCPoint4[17823] = {X 369.6229, Y 26.1959, Z -5.5000, A 0.000, B 0.000, C 0.000 }
gfCNCPoint4[17824] = {X 369.4629, Y 28.4279, Z -5.5000, A 0.000, B 0.000, C 0.000 }
gfCNCPoint4[17825] = {X 369.1452, Y 30.6430, Z -5.5000, A 0.000, B 0.000, C 0.000 }
gfCNCPoint4[17826] = {X 368.6474, Y 32.8845, Z -5.5000, A 0.000, B 0.000, C 0.000 }
gfCNCPoint4[17827] = {X 367.9414, Y 35.0695, Z -5.5000, A 0.000, B 0.000, C 0.000 }
gfCNCPoint4[17828] = {X 367.0333, Y 37.1785, Z -5.5000, A 0.000, B 0.000, C 0.000 }
gfCNCPoint4[17829] = {X 365.9313, Y 39.1929, Z -5.5000, A 0.000, B 0.000, C 0.000 }
gfCNCPoint4[17830] = {X 364.6449, Y 41.0950, Z -5.5000, A 0.000, B 0.000, C 0.000 }
gfCNCPoint4[17831] = {X 364.5295, Y 41.2530, Z -5.5000, A 0.000, B 0.000, C 0.000 }
gfCNCPoint4[17832] = {X 363.1396, Y 42.9173, Z -5.5000, A 0.000, B 0.000, C 0.000 }
gfCNCPoint4[17833] = {X 361.5913, Y 44.4354, Z -5.5000, A 0.000, B 0.000, C 0.000 }
gfCNCPoint4[17834] = {X 359.9001, Y 45.7925, Z -5.5000, A 0.000, B 0.000, C 0.000 }
gfCNCPoint4[17835] = {X 358.0826, Y 46.9750, Z -5.5000, A 0.000, B 0.000, C 0.000 }
gfCNCPoint4[17836] = {X 356.1567, Y 47.9713, Z -5.5000, A 0.000, B 0.000, C 0.000 }
gfCNCPoint4[17837] = {X 353.9741, Y 48.7857, Z -5.5000, A 0.000, B 0.000, C 0.000 }
gfCNCPoint4[17838] = {X 351.7199, Y 49.3739, Z -5.5000, A 0.000, B 0.000, C 0.000 }
gfCNCPoint4[17839] = {X 349.4176, Y 49.7296, Z -5.5000, A 0.000, B 0.000, C 0.000 }
gfCNCPoint4[17840] = {X 347.0911, Y 49.8493, Z -5.5000, A 0.000, B 0.000, C 0.000 }
gfCNCPoint4[17841] = {X 345.0383, Y 49.8148, Z -5.5000, A 0.000, B 0.000, C 0.000 }
gfCNCPoint4[17842] = {X 342.9962, Y 49.6024, Z -5.5000, A 0.000, B 0.000, C 0.000 }
gfCNCPoint4[17843] = {X 340.9803, Y 49.2138, Z -5.5000, A 0.000, B 0.000, C 0.000 }
gfCNCPoint4[17844] = {X 339.0056, Y 48.6517, Z -5.5000, A 0.000, B 0.000, C 0.000 }
gfCNCPoint4[17845] = {X 337.0872, Y 47.9205, Z -5.5000, A 0.000, B 0.000, C 0.000 }
gfCNCPoint4[17846] = {X 335.2394, Y 47.0256, Z -5.5000, A 0.000, B 0.000, C 0.000 }
gfCNCPoint4[17847] = {X 333.6458, Y 46.0411, Z -5.5000, A 0.000, B 0.000, C 0.000 }
gfCNCPoint4[17848] = {X 332.1352, Y 44.9334, Z -5.5000, A 0.000, B 0.000, C 0.000 }
gfCNCPoint4[17849] = {X 330.7172, Y 43.7094, Z -5.5000, A 0.000, B 0.000, C 0.000 }
gfCNCPoint4[17850] = {X 329.7930, Y 43.7230, Z -5.5000, A 0.000, B 0.000, C 0.000 }
gfCNCPoint4[17851] = {X 328.8887, Y 43.5322, Z -5.5000, A 0.000, B 0.000, C 0.000 }
gfCNCPoint4[17852] = {X 328.0488, Y 43.1464, Z -5.5000, A 0.000, B 0.000, C 0.000 }
gfCNCPoint4[17853] = {X 327.3148, Y 42.5847, Z -5.5000, A 0.000, B 0.000, C 0.000 }
gfCNCPoint4[17854] = {X 326.6925, Y 41.9780, Z -5.5000, A 0.000, B 0.000, C 0.000 }
gfCNCPoint4[17855] = {X 326.0873, Y 41.2331, Z -5.5000, A 0.000, B 0.000, C 0.000 }
gfCNCPoint4[17856] = {X 325.6690, Y 40.3693, Z -5.5000, A 0.000, B 0.000, C 0.000 }
gfCNCPoint4[17857] = {X 325.4597, Y 39.4326, Z -5.5000, A 0.000, B 0.000, C 0.000 }
gfCNCPoint4[17858] = {X 325.4707, Y 38.4730, Z -5.5000, A 0.000, B 0.000, C 0.000 }
gfCNCPoint4[17859] = {X 325.7013, Y 37.5413, Z -5.5000, A 0.000, B 0.000, C 0.000 }
gfCNCPoint4[17860] = {X 326.1392, Y 36.6874, Z -5.5000, A 0.000, B 0.000, C 0.000 }
gfCNCPoint4[17861] = {X 330.3725, Y 30.3576, Z -5.5000, A 0.000, B 0.000, C 0.000 }
gfCNCPoint4[17862] = {X 330.9517, Y 29.6673, Z -5.5000, A 0.000, B 0.000, C 0.000 }
gfCNCPoint4[17863] = {X 331.6658, Y 29.1179, Z -5.5000, A 0.000, B 0.000, C 0.000 }
gfCNCPoint4[17864] = {X 332.4816, Y 28.7351, Z -5.5000, A 0.000, B 0.000, C 0.000 }
gfCNCPoint4[17865] = {X 333.3606, Y 28.5369, Z -5.5000, A 0.000, B 0.000, C 0.000 }
gfCNCPoint4[17866] = {X 334.2616, Y 28.5327, Z -5.5000, A 0.000, B 0.000, C 0.000 }
gfCNCPoint4[17867] = {X 335.1425, Y 28.7227, Z -5.5000, A 0.000, B 0.000, C 0.000 }
gfCNCPoint4[17868] = {X 335.9617, Y 29.0978, Z -5.5000, A 0.000, B 0.000, C 0.000 }
gfCNCPoint4[17869] = {X 336.6810, Y 29.6405, Z -5.5000, A 0.000, B 0.000, C 0.000 }
gfCNCPoint4[17870] = {X 337.3163, Y 30.2523, Z -5.5000, A 0.000, B 0.000, C 0.000 }
gfCNCPoint4[17871] = {X 337.8307, Y 30.8657, Z -5.5000, A 0.000, B 0.000, C 0.000 }
gfCNCPoint4[17872] = {X 338.2181, Y 31.5663, Z -5.5000, A 0.000, B 0.000, C 0.000 }
gfCNCPoint4[17873] = {X 338.4641, Y 32.3281, Z -5.5000, A 0.000, B 0.000, C 0.000 }
gfCNCPoint4[17874] = {X 338.5597, Y 33.1230, Z -5.5000, A 0.000, B 0.000, C 0.000 }
gfCNCPoint4[17875] = {X 338.5012, Y 33.9214, Z -5.5000, A 0.000, B 0.000, C 0.000 }
gfCNCPoint4[17876] = {X 339.3030, Y 34.6466, Z -5.5000, A 0.000, B 0.000, C 0.000 }
gfCNCPoint4[17877] = {X 340.1367, Y 35.3350, Z -5.5000, A 0.000, B 0.000, C 0.000 }
gfCNCPoint4[17878] = {X 341.4534, Y 36.1993, Z -5.5000, A 0.000, B 0.000, C 0.000 }
gfCNCPoint4[17879] = {X 342.8819, Y 36.8625, Z -5.5000, A 0.000, B 0.000, C 0.000 }
gfCNCPoint4[17880] = {X 344.3917, Y 37.3105, Z -5.5000, A 0.000, B 0.000, C 0.000 }
gfCNCPoint4[17881] = {X 345.9508, Y 37.5338, Z -5.5000, A 0.000, B 0.000, C 0.000 }
gfCNCPoint4[17882] = {X 347.5257, Y 37.5276, Z -5.5000, A 0.000, B 0.000, C 0.000 }
gfCNCPoint4[17883] = {X 348.7016, Y 37.3894, Z -5.5000, A 0.000, B 0.000, C 0.000 }
gfCNCPoint4[17884] = {X 349.8494, Y 37.0989, Z -5.5000, A 0.000, B 0.000, C 0.000 }
gfCNCPoint4[17885] = {X 350.9495, Y 36.6611, Z -5.5000, A 0.000, B 0.000, C 0.000 }
gfCNCPoint4[17886] = {X 351.9831, Y 36.0835, Z -5.5000, A 0.000, B 0.000, C 0.000 }
gfCNCPoint4[17887] = {X 352.9325, Y 35.3760, Z -5.5000, A 0.000, B 0.000, C 0.000 }
gfCNCPoint4[17888] = {X 354.1011, Y 34.2407, Z -5.5000, A 0.000, B 0.000, C 0.000 }
gfCNCPoint4[17889] = {X 355.1123, Y 32.9634, Z -5.5000, A 0.000, B 0.000, C 0.000 }
gfCNCPoint4[17890] = {X 355.9492, Y 31.5655, Z -5.5000, A 0.000, B 0.000, C 0.000 }
gfCNCPoint4[17891] = {X 356.5975, Y 30.0708, Z -5.5000, A 0.000, B 0.000, C 0.000 }
gfCNCPoint4[17892] = {X 357.0463, Y 28.5046, Z -5.5000, A 0.000, B 0.000, C 0.000 }
gfCNCPoint4[17893] = {X 357.3220, Y 26.8012, Z -5.5000, A 0.000, B 0.000, C 0.000 }
gfCNCPoint4[17894] = {X 357.4343, Y 25.0793, Z -5.5000, A 0.000, B 0.000, C 0.000 }
gfCNCPoint4[17895] = {X 357.3822, Y 23.3545, Z -5.5000, A 0.000, B 0.000, C 0.000 }
gfCNCPoint4[17896] = {X 357.1662, Y 21.6425, Z -5.5000, A 0.000, B 0.000, C 0.000 }
gfCNCPoint4[17897] = {X 356.8075, Y 20.1065, Z -5.5000, A 0.000, B 0.000, C 0.000 }
gfCNCPoint4[17898] = {X 356.2504, Y 18.6308, Z -5.5000, A 0.000, B 0.000, C 0.000 }
gfCNCPoint4[17899] = {X 355.5045, Y 17.2409, Z -5.5000, A 0.000, B 0.000, C 0.000 }
gfCNCPoint4[17900] = {X 354.5828, Y 15.9608, Z -5.5000, A 0.000, B 0.000, C 0.000 }
gfCNCPoint4[17901] = {X 353.6970, Y 15.0178, Z -5.5000, A 0.000, B 0.000, C 0.000 }
gfCNCPoint4[17902] = {X 352.6889, Y 14.2068, Z -5.5000, A 0.000, B 0.000, C 0.000 }
gfCNCPoint4[17903] = {X 351.5782, Y 13.5433, Z -5.5000, A 0.000, B 0.000, C 0.000 }
gfCNCPoint4[17904] = {X 350.3862, Y 13.0403, Z -5.5000, A 0.000, B 0.000, C 0.000 }
gfCNCPoint4[17905] = {X 349.1360, Y 12.7073, Z -5.5000, A 0.000, B 0.000, C 0.000 }
gfCNCPoint4[17906] = {X 347.5978, Y 12.5019, Z -5.5000, A 0.000, B 0.000, C 0.000 }
gfCNCPoint4[17907] = {X 346.0462, Y 12.4738, Z -5.5000, A 0.000, B 0.000, C 0.000 }
gfCNCPoint4[17908] = {X 344.5015, Y 12.6234, Z -5.5000, A 0.000, B 0.000, C 0.000 }
gfCNCPoint4[17909] = {X 342.9841, Y 12.9488, Z -5.5000, A 0.000, B 0.000, C 0.000 }
gfCNCPoint4[17910] = {X 341.5139, Y 13.4457, Z -5.5000, A 0.000, B 0.000, C 0.000 }
gfCNCPoint4[17911] = {X 340.1102, Y 14.1075, Z -5.5000, A 0.000, B 0.000, C 0.000 }
gfCNCPoint4[17912] = {X 338.7915, Y 14.9255, Z -5.5000, A 0.000, B 0.000, C 0.000 }
gfCNCPoint4[17913] = {X 338.7691, Y 15.7571, Z -5.5000, A 0.000, B 0.000, C 0.000 }
gfCNCPoint4[17914] = {X 338.5817, Y 16.5676, Z -5.5000, A 0.000, B 0.000, C 0.000 }
gfCNCPoint4[17915] = {X 338.2368, Y 17.3246, Z -5.5000, A 0.000, B 0.000, C 0.000 }
gfCNCPoint4[17916] = {X 337.7481, Y 17.9978, Z -5.5000, A 0.000, B 0.000, C 0.000 }
gfCNCPoint4[17917] = {X 337.1353, Y 18.5604, Z -5.5000, A 0.000, B 0.000, C 0.000 }
gfCNCPoint4[17918] = {X 336.4209, Y 19.0861, Z -5.5000, A 0.000, B 0.000, C 0.000 }
gfCNCPoint4[17919] = {X 335.6353, Y 19.5283, Z -5.5000, A 0.000, B 0.000, C 0.000 }
gfCNCPoint4[17920] = {X 334.7729, Y 19.7908, Z -5.5000, A 0.000, B 0.000, C 0.000 }
gfCNCPoint4[17921] = {X 333.8742, Y 19.8614, Z -5.5000, A 0.000, B 0.000, C 0.000 }
gfCNCPoint4[17922] = {X 332.9814, Y 19.7367, Z -5.5000, A 0.000, B 0.000, C 0.000 }
gfCNCPoint4[17923] = {X 332.1364, Y 19.4226, Z -5.5000, A 0.000, B 0.000, C 0.000 }
gfCNCPoint4[17924] = {X 331.3789, Y 18.9339, Z -5.5000, A 0.000, B 0.000, C 0.000 }
gfCNCPoint4[17925] = {X 330.7445, Y 18.2934, Z -5.5000, A 0.000, B 0.000, C 0.000 }
gfCNCPoint4[17926] = {X 330.2630, Y 17.5314, Z -5.5000, A 0.000, B 0.000, C 0.000 }
gfCNCPoint4[17927] = {X 326.7381, Y 10.2803, Z -5.5000, A 0.000, B 0.000, C 0.000 }
gfCNCPoint4[17928] = {X 326.4156, Y 9.3505, Z -5.5000, A 0.000, B 0.000, C 0.000 }
gfCNCPoint4[17929] = {X 326.3205, Y 8.3711, Z -5.5000, A 0.000, B 0.000, C 0.000 }
gfCNCPoint4[17930] = {X 326.4581, Y 7.3967, Z -5.5000, A 0.000, B 0.000, C 0.000 }
gfCNCPoint4[17931] = {X 326.8207, Y 6.4819, Z -5.5000, A 0.000, B 0.000, C 0.000 }
gfCNCPoint4[17932] = {X 327.3881, Y 5.6778, Z -5.5000, A 0.000, B 0.000, C 0.000 }
gfCNCPoint4[17933] = {X 328.1285, Y 5.0296, Z -5.5000, A 0.000, B 0.000, C 0.000 }
gfCNCPoint4[17934] = {X 328.7983, Y 4.5709, Z -5.5000, A 0.000, B 0.000, C 0.000 }
gfCNCPoint4[17935] = {X 329.6632, Y 4.1254, Z -5.5000, A 0.000, B 0.000, C 0.000 }
gfCNCPoint4[17936] = {X 330.6079, Y 3.8929, Z -5.5000, A 0.000, B 0.000, C 0.000 }
gfCNCPoint4[17937] = {X 331.5808, Y 3.8863, Z -5.5000, A 0.000, B 0.000, C 0.000 }
gfCNCPoint4[17938] = {X 332.5287, Y 4.1058, Z -5.5000, A 0.000, B 0.000, C 0.000 }
gfCNCPoint4[17939] = {X 334.0385, Y 3.2593, Z -5.5000, A 0.000, B 0.000, C 0.000 }
gfCNCPoint4[17940] = {X 335.5974, Y 2.5071, Z -5.5000, A 0.000, B 0.000, C 0.000 }
gfCNCPoint4[17941] = {X 337.7207, Y 1.6457, Z -5.5000, A 0.000, B 0.000, C 0.000 }
gfCNCPoint4[17942] = {X 339.9113, Y 0.9736, Z -5.5000, A 0.000, B 0.000, C 0.000 }
gfCNCPoint4[17943] = {X 342.1523, Y 0.4962, Z -5.5000, A 0.000, B 0.000, C 0.000 }
gfCNCPoint4[17944] = {X 344.4266, Y 0.2169, Z -5.5000, A 0.000, B 0.000, C 0.000 }
gfCNCPoint4[17945] = {X 346.7166, Y 0.1381, Z -5.5000, A 0.000, B 0.000, C 0.000 }
gfCNCPoint4[17946] = {X 349.0046, Y 0.2602, Z -5.5000, A 0.000, B 0.000, C 0.000 }
gfCNCPoint4[17947] = {X 351.2732, Y 0.5824, Z -5.5000, A 0.000, B 0.000, C 0.000 }
gfCNCPoint4[17948] = {X 351.5571, Y 0.6355, Z -5.5000, A 0.000, B 0.000, C 0.000 }
gfCNCPoint4[17949] = {X 352.2921, Y -3.2964, Z -5.5000, A 0.000, B 0.000, C 0.000 }
gfCNCPoint4[17950] = {X 351.5424, Y 0.7141, Z -5.5000, A 0.000, B 0.000, C 0.000 }
gfCNCPoint4[17951] = {X 351.8247, Y 0.7669, Z -5.5000, A 0.000, B 0.000, C 0.000 }
gfCNCPoint4[17952] = {X 353.7527, Y 1.2519, Z -5.5000, A 0.000, B 0.000, C 0.000 }
gfCNCPoint4[17953] = {X 355.6255, Y 1.9191, Z -5.5000, A 0.000, B 0.000, C 0.000 }
gfCNCPoint4[17954] = {X 357.4260, Y 2.7621, Z -5.5000, A 0.000, B 0.000, C 0.000 }
gfCNCPoint4[17955] = {X 359.1377, Y 3.7734, Z -5.5000, A 0.000, B 0.000, C 0.000 }
gfCNCPoint4[17956] = {X 360.7449, Y 4.9437, Z -5.5000, A 0.000, B 0.000, C 0.000 }
gfCNCPoint4[17957] = {X 362.2328, Y 6.2622, Z -5.5000, A 0.000, B 0.000, C 0.000 }
gfCNCPoint4[17958] = {X 363.5879, Y 7.7169, Z -5.5000, A 0.000, B 0.000, C 0.000 }
gfCNCPoint4[17959] = {X 364.9262, Y 9.4565, Z -5.5000, A 0.000, B 0.000, C 0.000 }
gfCNCPoint4[17960] = {X 366.1058, Y 11.3074, Z -5.5000, A 0.000, B 0.000, C 0.000 }
gfCNCPoint4[17961] = {X 367.1176, Y 13.2551, Z -5.5000, A 0.000, B 0.000, C 0.000 }
gfCNCPoint4[17962] = {X 367.9536, Y 15.2844, Z -5.5000, A 0.000, B 0.000, C 0.000 }
gfCNCPoint4[17963] = {X 368.6074, Y 17.3796, Z -5.5000, A 0.000, B 0.000, C 0.000 }
gfCNCPoint4[17964] = {X 369.0739, Y 19.5242, Z -5.5000, A 0.000, B 0.000, C 0.000 }
gfCNCPoint4[17965] = {X 369.3878, Y 21.7342, Z -5.5000, A 0.000, B 0.000, C 0.000 }
gfCNCPoint4[17966] = {X 369.5445, Y 23.9609, Z -5.5000, A 0.000, B 0.000, C 0.000 }
gfCNCPoint4[17967] = {X 369.5430, Y 26.1930, Z -5.5000, A 0.000, B 0.000, C 0.000 }
gfCNCPoint4[17968] = {X 369.3833, Y 28.4195, Z -5.5000, A 0.000, B 0.000, C 0.000 }
gfCNCPoint4[17969] = {X 369.0664, Y 30.6290, Z -5.5000, A 0.000, B 0.000, C 0.000 }
gfCNCPoint4[17970] = {X 368.5703, Y 32.8634, Z -5.5000, A 0.000, B 0.000, C 0.000 }
gfCNCPoint4[17971] = {X 367.8665, Y 35.0413, Z -5.5000, A 0.000, B 0.000, C 0.000 }
gfCNCPoint4[17972] = {X 366.9614, Y 37.1435, Z -5.5000, A 0.000, B 0.000, C 0.000 }
gfCNCPoint4[17973] = {X 365.8628, Y 39.1515, Z -5.5000, A 0.000, B 0.000, C 0.000 }
gfCNCPoint4[17974] = {X 364.5806, Y 41.0474, Z -5.5000, A 0.000, B 0.000, C 0.000 }
gfCNCPoint4[17975] = {X 364.4653, Y 41.2053, Z -5.5000, A 0.000, B 0.000, C 0.000 }
gfCNCPoint4[17976] = {X 363.0806, Y 42.8633, Z -5.5000, A 0.000, B 0.000, C 0.000 }
gfCNCPoint4[17977] = {X 361.5382, Y 44.3756, Z -5.5000, A 0.000, B 0.000, C 0.000 }
gfCNCPoint4[17978] = {X 359.8534, Y 45.7275, Z -5.5000, A 0.000, B 0.000, C 0.000 }
gfCNCPoint4[17979] = {X 358.0428, Y 46.9056, Z -5.5000, A 0.000, B 0.000, C 0.000 }
gfCNCPoint4[17980] = {X 356.1242, Y 47.8982, Z -5.5000, A 0.000, B 0.000, C 0.000 }
gfCNCPoint4[17981] = {X 353.9491, Y 48.7097, Z -5.5000, A 0.000, B 0.000, C 0.000 }
gfCNCPoint4[17982] = {X 351.7028, Y 49.2957, Z -5.5000, A 0.000, B 0.000, C 0.000 }
gfCNCPoint4[17983] = {X 349.4085, Y 49.6502, Z -5.5000, A 0.000, B 0.000, C 0.000 }
gfCNCPoint4[17984] = {X 347.0900, Y 49.7693, Z -5.5000, A 0.000, B 0.000, C 0.000 }
gfCNCPoint4[17985] = {X 345.0441, Y 49.7350, Z -5.5000, A 0.000, B 0.000, C 0.000 }
gfCNCPoint4[17986] = {X 343.0089, Y 49.5235, Z -5.5000, A 0.000, B 0.000, C 0.000 }
gfCNCPoint4[17987] = {X 340.9997, Y 49.1362, Z -5.5000, A 0.000, B 0.000, C 0.000 }
gfCNCPoint4[17988] = {X 339.0317, Y 48.5760, Z -5.5000, A 0.000, B 0.000, C 0.000 }
gfCNCPoint4[17989] = {X 337.1197, Y 47.8474, Z -5.5000, A 0.000, B 0.000, C 0.000 }
gfCNCPoint4[17990] = {X 335.2780, Y 46.9556, Z -5.5000, A 0.000, B 0.000, C 0.000 }
gfCNCPoint4[17991] = {X 333.6796, Y 45.9675, Z -5.5000, A 0.000, B 0.000, C 0.000 }
gfCNCPoint4[17992] = {X 332.1652, Y 44.8550, Z -5.5000, A 0.000, B 0.000, C 0.000 }
gfCNCPoint4[17993] = {X 330.7443, Y 43.6252, Z -5.5000, A 0.000, B 0.000, C 0.000 }
gfCNCPoint4[17994] = {X 329.8287, Y 43.6460, Z -5.5000, A 0.000, B 0.000, C 0.000 }
gfCNCPoint4[17995] = {X 328.9316, Y 43.4621, Z -5.5000, A 0.000, B 0.000, C 0.000 }
gfCNCPoint4[17996] = {X 328.0980, Y 43.0827, Z -5.5000, A 0.000, B 0.000, C 0.000 }
gfCNCPoint4[17997] = {X 327.3701, Y 42.5270, Z -5.5000, A 0.000, B 0.000, C 0.000 }
gfCNCPoint4[17998] = {X 326.7483, Y 41.9207, Z -5.5000, A 0.000, B 0.000, C 0.000 }
gfCNCPoint4[17999] = {X 326.1548, Y 41.1901, Z -5.5000, A 0.000, B 0.000, C 0.000 }
gfCNCPoint4[18000] = {X 325.7445, Y 40.3430, Z -5.5000, A 0.000, B 0.000, C 0.000 }
gfCNCPoint4[18001] = {X 325.5393, Y 39.4243, Z -5.5000, A 0.000, B 0.000, C 0.000 }
gfCNCPoint4[18002] = {X 325.5500, Y 38.4831, Z -5.5000, A 0.000, B 0.000, C 0.000 }
gfCNCPoint4[18003] = {X 325.7762, Y 37.5694, Z -5.5000, A 0.000, B 0.000, C 0.000 }
gfCNCPoint4[18004] = {X 326.2057, Y 36.7318, Z -5.5000, A 0.000, B 0.000, C 0.000 }
gfCNCPoint4[18005] = {X 330.4390, Y 30.4021, Z -5.5000, A 0.000, B 0.000, C 0.000 }
gfCNCPoint4[18006] = {X 331.0070, Y 29.7251, Z -5.5000, A 0.000, B 0.000, C 0.000 }
gfCNCPoint4[18007] = {X 331.7074, Y 29.1862, Z -5.5000, A 0.000, B 0.000, C 0.000 }
gfCNCPoint4[18008] = {X 332.5073, Y 28.8108, Z -5.5000, A 0.000, B 0.000, C 0.000 }
gfCNCPoint4[18009] = {X 333.3694, Y 28.6165, Z -5.5000, A 0.000, B 0.000, C 0.000 }
gfCNCPoint4[18010] = {X 334.2531, Y 28.6123, Z -5.5000, A 0.000, B 0.000, C 0.000 }
gfCNCPoint4[18011] = {X 335.1169, Y 28.7985, Z -5.5000, A 0.000, B 0.000, C 0.000 }
gfCNCPoint4[18012] = {X 335.9204, Y 29.1663, Z -5.5000, A 0.000, B 0.000, C 0.000 }
gfCNCPoint4[18013] = {X 336.6259, Y 29.6985, Z -5.5000, A 0.000, B 0.000, C 0.000 }
gfCNCPoint4[18014] = {X 337.2602, Y 30.3094, Z -5.5000, A 0.000, B 0.000, C 0.000 }
gfCNCPoint4[18015] = {X 337.7696, Y 30.9180, Z -5.5000, A 0.000, B 0.000, C 0.000 }
gfCNCPoint4[18016] = {X 338.1514, Y 31.6138, Z -5.5000, A 0.000, B 0.000, C 0.000 }
gfCNCPoint4[18017] = {X 338.3914, Y 32.3703, Z -5.5000, A 0.000, B 0.000, C 0.000 }
gfCNCPoint4[18018] = {X 338.4804, Y 33.1589, Z -5.5000, A 0.000, B 0.000, C 0.000 }
gfCNCPoint4[18019] = {X 338.4150, Y 33.9499, Z -5.5000, A 0.000, B 0.000, C 0.000 }
gfCNCPoint4[18020] = {X 339.2346, Y 34.6933, Z -5.5000, A 0.000, B 0.000, C 0.000 }
gfCNCPoint4[18021] = {X 340.0877, Y 35.3982, Z -5.5000, A 0.000, B 0.000, C 0.000 }
gfCNCPoint4[18022] = {X 341.4139, Y 36.2689, Z -5.5000, A 0.000, B 0.000, C 0.000 }
gfCNCPoint4[18023] = {X 342.8529, Y 36.9371, Z -5.5000, A 0.000, B 0.000, C 0.000 }
gfCNCPoint4[18024] = {X 344.3738, Y 37.3885, Z -5.5000, A 0.000, B 0.000, C 0.000 }
gfCNCPoint4[18025] = {X 345.9443, Y 37.6136, Z -5.5000, A 0.000, B 0.000, C 0.000 }
gfCNCPoint4[18026] = {X 347.5308, Y 37.6075, Z -5.5000, A 0.000, B 0.000, C 0.000 }
gfCNCPoint4[18027] = {X 348.7169, Y 37.4679, Z -5.5000, A 0.000, B 0.000, C 0.000 }
gfCNCPoint4[18028] = {X 349.8747, Y 37.1748, Z -5.5000, A 0.000, B 0.000, C 0.000 }
gfCNCPoint4[18029] = {X 350.9843, Y 36.7332, Z -5.5000, A 0.000, B 0.000, C 0.000 }
gfCNCPoint4[18030] = {X 352.0268, Y 36.1506, Z -5.5000, A 0.000, B 0.000, C 0.000 }
gfCNCPoint4[18031] = {X 352.9844, Y 35.4369, Z -5.5000, A 0.000, B 0.000, C 0.000 }
gfCNCPoint4[18032] = {X 354.1604, Y 34.2943, Z -5.5000, A 0.000, B 0.000, C 0.000 }
gfCNCPoint4[18033] = {X 355.1782, Y 33.0088, Z -5.5000, A 0.000, B 0.000, C 0.000 }
gfCNCPoint4[18034] = {X 356.0204, Y 31.6019, Z -5.5000, A 0.000, B 0.000, C 0.000 }
gfCNCPoint4[18035] = {X 356.6729, Y 30.0976, Z -5.5000, A 0.000, B 0.000, C 0.000 }
gfCNCPoint4[18036] = {X 357.1245, Y 28.5214, Z -5.5000, A 0.000, B 0.000, C 0.000 }
